    movel(pose_trans(stn7_plane, pose_trans(p[.109811488584, -1.023382701287, -.166619380160, .003048702642, -.008599620441, 2.442192581404], stn7_dr1_dwn_p_p)), a=0.1, v=0.05)
    # begin: URCap Program Node
    #   Source: Robotiq_Grippers, 1.8.13.22852, Robotiq Inc.
    #   Type: Greifer
    $ 1330 "Greifer offen (1)"
    if not(gripper_connected[0]):
      popup("Greifer 1 muss verbunden sein, um dieses Programm auszuführen.", "Keine Verbindung", False, True, True)
    end
    if not(rq_is_gripper_activated("1")):
      popup("Greifer 1 ist nicht aktiviert. Wechseln Sie zur Registerkarte Installation > Greifer, um ihn zu aktivieren und das Programm erneut auszuführen.", "Nicht aktiviert", False, True, True)
    end
    rq_set_pos_spd_for(0, 255, 0, "1")
    rq_wait_pos_spe_for_request(0, 255, 0, "1")
    rq_go_to("1")
    rq_wait("1")
    # end: URCap Program Node
    $ 1331 "stn7_dr1_up_p" "breakAfter"
    set_tcp(p[-3.0E-4,2.5E-4,0.1575,0.0,0.0,0.0])
    movel(pose_trans(stn7_plane, pose_trans(p[.109811488584, -1.023382701287, -.166619380160, .003048702642, -.008599620441, 2.442192581404], stn7_dr1_up_p_p)), a=0.1, v=0.05)
    # begin: URCap Program Node
    #   Source: Robotiq_Grippers, 1.8.13.22852, Robotiq Inc.
    #   Type: Greifer
    $ 1332 "Greifer geschlossen (1)"
    if not(gripper_connected[0]):
      popup("Greifer 1 muss verbunden sein, um dieses Programm auszuführen.", "Keine Verbindung", False, True, True)
    end
    if not(rq_is_gripper_activated("1")):
      popup("Greifer 1 ist nicht aktiviert. Wechseln Sie zur Registerkarte Installation > Greifer, um ihn zu aktivieren und das Programm erneut auszuführen.", "Nicht aktiviert", False, True, True)
    end
    rq_set_pos_spd_for(255, 255, 0, "1")
    rq_wait_pos_spe_for_request(255, 255, 0, "1")
    rq_go_to("1")
    rq_wait("1")
    # end: URCap Program Node
    $ 1333 "FahreAchse"
    $ 1334 "stn7_ld_apr_p" "breakAfter"
    set_tcp(p[-3.0E-4,2.5E-4,0.1575,0.0,0.0,0.0])
    movej(get_inverse_kin(pose_trans(stn7_plane, pose_trans(p[.109811488584, -1.023382701287, -.166619380160, .003048702642, -.008599620441, 2.442192581404], stn7_ld_apr_p_p)), qnear=stn7_ld_apr_p_q), a=2.443460952792061, v=1.7453292519943295)
    $ 1335 "FahreLinear"
    $ 1336 "stn7_ld_press_p" "breakAfter"
    set_tcp(p[-3.0E-4,2.5E-4,0.1575,0.0,0.0,0.0])
    movel(pose_trans(stn7_plane, pose_trans(p[.109811488584, -1.023382701287, -.166619380160, .003048702642, -.008599620441, 2.442192581404], stn7_ld_press_p_p)), a=0.6, v=0.1)
    $ 1337 "Warten: 1.0"
    sleep(1.0)
    $ 1338 "stn7_ld_apr_p" "breakAfter"
    set_tcp(p[-3.0E-4,2.5E-4,0.1575,0.0,0.0,0.0])
    movel(pose_trans(stn7_plane, pose_trans(p[.109811488584, -1.023382701287, -.166619380160, .003048702642, -.008599620441, 2.442192581404], stn7_ld_apr_p_p)), a=0.6, v=0.1)
    $ 1339 "qMast.set_init_alarm(7)"
    qMast.set_init_alarm(7)
    $ 1340 "FahreAchse"
    $ 1341 "stn7_home_p" "breakAfter"
    set_tcp(p[-3.0E-4,2.5E-4,0.1575,0.0,0.0,0.0])
    movej(get_inverse_kin(pose_trans(stn7_plane, pose_trans(p[.109811488584, -1.023382701287, -.166619380160, .003048702642, -.008599620441, 2.442192581404], stn7_home_p_p)), qnear=stn7_home_p_q), a=1.3962634015954636, v=1.0471975511965976)
  end
  def stn7_open_doors():
    $ 1342 "stn7_open_doors" "noBreak"
    $ 1343 "FahreAchse"
    $ 1345 "stn7_retrct1_p" "breakAfter"
    set_tcp(p[-3.0E-4,2.5E-4,0.1575,0.0,0.0,0.0])
    movej(get_inverse_kin(pose_trans(stn7_plane, pose_trans(p[.109811488584, -1.023382701287, -.166619380160, .003048702642, -.008599620441, 2.442192581404], stn7_retrct1_p_p)), qnear=stn7_retrct1_p_q), a=1.3962634015954636, v=1.0471975511965976)
    $ 1346 "stn7_dr1_up_p" "breakAfter"
    set_tcp(p[-3.0E-4,2.5E-4,0.1575,0.0,0.0,0.0])
    movej(get_inverse_kin(pose_trans(stn7_plane, pose_trans(p[.109811488584, -1.023382701287, -.166619380160, .003048702642, -.008599620441, 2.442192581404], stn7_dr1_up_p_p)), qnear=stn7_dr1_up_p_q), a=1.3962634015954636, v=1.0471975511965976)
    # begin: URCap Program Node
    #   Source: Robotiq_Grippers, 1.8.13.22852, Robotiq Inc.
    #   Type: Greifer
    $ 1347 "Greifer offen (1)"
    if not(gripper_connected[0]):
      popup("Greifer 1 muss verbunden sein, um dieses Programm auszuführen.", "Keine Verbindung", False, True, True)
    end
    if not(rq_is_gripper_activated("1")):
      popup("Greifer 1 ist nicht aktiviert. Wechseln Sie zur Registerkarte Installation > Greifer, um ihn zu aktivieren und das Programm erneut auszuführen.", "Nicht aktiviert", False, True, True)
    end
    rq_set_pos_spd_for(0, 255, 0, "1")
    rq_wait_pos_spe_for_request(0, 255, 0, "1")
    rq_go_to("1")
    rq_wait("1")
    # end: URCap Program Node
    $ 1348 "FahreLinear"
    $ 1349 "stn7_dr1_dwn_p" "breakAfter"
    set_tcp(p[-3.0E-4,2.5E-4,0.1575,0.0,0.0,0.0])
    movel(pose_trans(stn7_plane, pose_trans(p[.109811488584, -1.023382701287, -.166619380160, .003048702642, -.008599620441, 2.442192581404], stn7_dr1_dwn_p_p)), a=0.3, v=0.1)
    $ 1350 "stn7_dr1_open_p" "breakAfter"
    set_tcp(p[-3.0E-4,2.5E-4,0.1575,0.0,0.0,0.0])
    movel(pose_trans(stn7_plane, pose_trans(p[.109811488584, -1.023382701287, -.166619380160, .003048702642, -.008599620441, 2.442192581404], stn7_dr1_open_p_p)), a=0.3, v=0.1)
    $ 1351 "stn7_dr2_ohp1_p" "breakAfter"
    set_tcp(p[-3.0E-4,2.5E-4,0.1575,0.0,0.0,0.0])
    movel(pose_trans(stn7_plane, pose_trans(p[.109811488584, -1.023382701287, -.166619380160, .003048702642, -.008599620441, 2.442192581404], stn7_dr2_ohp1_p_p)), a=0.3, v=0.1)
    $ 1352 "FahreLinear"
    $ 1353 "stn7_dr2_up_p" "breakAfter"
    set_tcp(p[-3.0E-4,2.5E-4,0.1575,0.0,0.0,0.0])
    movel(pose_trans(stn7_plane, pose_trans(p[.109811488584, -1.023382701287, -.166619380160, .003048702642, -.008599620441, 2.442192581404], stn7_dr2_up_p_p)), a=0.3, v=0.1)
    $ 1354 "stn7_dr2_dwn_p" "breakAfter"
    set_tcp(p[-3.0E-4,2.5E-4,0.1575,0.0,0.0,0.0])
    movel(pose_trans(stn7_plane, pose_trans(p[.109811488584, -1.023382701287, -.166619380160, .003048702642, -.008599620441, 2.442192581404], stn7_dr2_dwn_p_p)), a=0.3, v=0.1)
    $ 1355 "stn7_dr2_open_p" "breakAfter"
    set_tcp(p[-3.0E-4,2.5E-4,0.1575,0.0,0.0,0.0])
    movel(pose_trans(stn7_plane, pose_trans(p[.109811488584, -1.023382701287, -.166619380160, .003048702642, -.008599620441, 2.442192581404], stn7_dr2_open_p_p)), a=0.3, v=0.1)
    $ 1356 "stn7_dr2_ohp1_p" "breakAfter"
    set_tcp(p[-3.0E-4,2.5E-4,0.1575,0.0,0.0,0.0])
    movel(pose_trans(stn7_plane, pose_trans(p[.109811488584, -1.023382701287, -.166619380160, .003048702642, -.008599620441, 2.442192581404], stn7_dr2_ohp1_p_p)), a=0.3, v=0.1)
    # begin: URCap Program Node
    #   Source: Robotiq_Grippers, 1.8.13.22852, Robotiq Inc.
    #   Type: Greifer
    $ 1357 "Greifer geschlossen (1)"
    if not(gripper_connected[0]):
      popup("Greifer 1 muss verbunden sein, um dieses Programm auszuführen.", "Keine Verbindung", False, True, True)
    end
    if not(rq_is_gripper_activated("1")):
      popup("Greifer 1 ist nicht aktiviert. Wechseln Sie zur Registerkarte Installation > Greifer, um ihn zu aktivieren und das Programm erneut auszuführen.", "Nicht aktiviert", False, True, True)
    end
    rq_set_pos_spd_for(255, 255, 0, "1")
    rq_wait_pos_spe_for_request(255, 255, 0, "1")
    rq_go_to("1")
    rq_wait("1")
    # end: URCap Program Node
    $ 1358 "FahreAchse"
    $ 1359 "stn7_home_p" "breakAfter"
    set_tcp(p[-3.0E-4,2.5E-4,0.1575,0.0,0.0,0.0])
    movej(get_inverse_kin(pose_trans(stn7_plane, pose_trans(p[.109811488584, -1.023382701287, -.166619380160, .003048702642, -.008599620441, 2.442192581404], stn7_home_p_p)), qnear=stn7_home_p_q), a=1.3962634015954636, v=1.0471975511965976)
  end
  def stn7_close_doors():
    $ 1360 "stn7_close_doors" "noBreak"
    # begin: URCap Program Node
    #   Source: Robotiq_Grippers, 1.8.13.22852, Robotiq Inc.
    #   Type: Greifer
    $ 1361 "Greifer geschlossen (1)"
    if not(gripper_connected[0]):
      popup("Greifer 1 muss verbunden sein, um dieses Programm auszuführen.", "Keine Verbindung", False, True, True)
    end
    if not(rq_is_gripper_activated("1")):
      popup("Greifer 1 ist nicht aktiviert. Wechseln Sie zur Registerkarte Installation > Greifer, um ihn zu aktivieren und das Programm erneut auszuführen.", "Nicht aktiviert", False, True, True)
    end
    rq_set_pos_spd_for(255, 128, 255, "1")
    rq_wait_pos_spe_for_request(255, 128, 255, "1")
    rq_go_to("1")
    rq_wait("1")
    # end: URCap Program Node
    $ 1362 "FahreAchse"
    $ 1363 "stn7_home_p" "breakAfter"
    set_tcp(p[-3.0E-4,2.5E-4,0.1575,0.0,0.0,0.0])
    movej(get_inverse_kin(pose_trans(stn7_plane, pose_trans(p[.109811488584, -1.023382701287, -.166619380160, .003048702642, -.008599620441, 2.442192581404], stn7_home_p_p)), qnear=stn7_home_p_q), a=1.3962634015954636, v=1.0471975511965976, r=0.1)
    $ 1364 "stn7_apr1_p" "breakAfter"
    set_tcp(p[-3.0E-4,2.5E-4,0.1575,0.0,0.0,0.0])
    movej(get_inverse_kin(pose_trans(stn7_plane, pose_trans(p[.109811488584, -1.023382701287, -.166619380160, .003048702642, -.008599620441, 2.442192581404], stn7_apr1_p_p)), qnear=stn7_apr1_p_q), a=1.3962634015954636, v=1.0471975511965976)
    $ 1365 "FahreLinear"
    $ 1366 "stn7_push1_p" "breakAfter"
    set_tcp(p[-3.0E-4,2.5E-4,0.1575,0.0,0.0,0.0])
    movel(pose_trans(stn7_plane, pose_trans(p[.109811488584, -1.023382701287, -.166619380160, .003048702642, -.008599620441, 2.442192581404], stn7_push1_p_p)), a=0.5, v=0.1)
    $ 1367 "stn7_apr1_p" "breakAfter"
    set_tcp(p[-3.0E-4,2.5E-4,0.1575,0.0,0.0,0.0])
    movel(pose_trans(stn7_plane, pose_trans(p[.109811488584, -1.023382701287, -.166619380160, .003048702642, -.008599620441, 2.442192581404], stn7_apr1_p_p)), a=1.2, v=0.25)
    $ 1368 "stn7_apr2_p" "breakAfter"
    set_tcp(p[-3.0E-4,2.5E-4,0.1575,0.0,0.0,0.0])
    movel(pose_trans(stn7_plane, pose_trans(p[.109811488584, -1.023382701287, -.166619380160, .003048702642, -.008599620441, 2.442192581404], stn7_apr2_p_p)), a=1.2, v=0.25)
    $ 1369 "stn7_push2_p" "breakAfter"
    set_tcp(p[-3.0E-4,2.5E-4,0.1575,0.0,0.0,0.0])
    movel(pose_trans(stn7_plane, pose_trans(p[.109811488584, -1.023382701287, -.166619380160, .003048702642, -.008599620441, 2.442192581404], stn7_push2_p_p)), a=0.5, v=0.1)
    $ 1370 "stn7_dr2_bk_p" "breakAfter"
    set_tcp(p[-3.0E-4,2.5E-4,0.1575,0.0,0.0,0.0])
    movel(pose_trans(stn7_plane, pose_trans(p[.109811488584, -1.023382701287, -.166619380160, .003048702642, -.008599620441, 2.442192581404], stn7_dr2_bk_p_p)), a=1.2, v=0.25)
  end
  def stn7_check_doors():
    $ 1371 "stn7_check_doors" "noBreak"
    $ 1372 "Schleife"
    while (True):
      $ 1373 "stn7_door_1_ok≔get_digital_in(2)"
      global stn7_door_1_ok=get_digital_in(2)
      $ 1374 "If stn7_door_1_ok ≟  False "
      if (stn7_door_1_ok  ==    False  ):
        $ 1376 "Meldung"
        popup(str_cat("",stn7_skype_msg), "Fehler", False, True, blocking=False)
        halt
      else:
        $ 1377 "Else" "noBreak"
        $ 1378 "stn7_door_2_ok≔get_digital_in(0)"
        global stn7_door_2_ok=get_digital_in(0)
        $ 1379 "If stn7_door_2_ok ≟  False "
        if (stn7_door_2_ok  ==    False  ):
          $ 1381 "Meldung"
          popup(str_cat("",stn7_skype_msg), "Fehler", False, True, blocking=False)
          halt
        else:
          $ 1382 "Else" "noBreak"
          $ 1383 "break"
          break
        end
      end
    end
  end
  def stn9_decap():
    $ 1384 "stn9_decap" "noBreak"
    $ 1385 "FahreAchse"
    $ 1386 "stn9_dcap_apr_p" "breakAfter"
    set_tcp(p[-3.0E-4,2.5E-4,0.1575,0.0,0.0,0.0])
    movej(get_inverse_kin(pose_trans(stn6_plane, pose_trans(p[.776557109756, -.878329076792, .250244777977, -.001605684562, .009314448336, 1.565629725105], stn9_dcap_apr_p_p)), qnear=stn9_dcap_apr_p_q), a=2.792526803190927, v=2.0943951023931953)
    $ 1387 "Einstellen Decap=Ein"
    set_standard_digital_out(2, True)
    $ 1388 "FahreLinear"
    $ 1389 "stn9_lv_tb_p" "breakAfter"
    set_tcp(p[-3.0E-4,2.5E-4,0.1575,0.0,0.0,0.0])
    movel(pose_trans(stn6_plane, pose_trans(p[.776557109756, -.878329076792, .250244777977, -.001605684562, .009314448336, 1.565629725105], stn9_lv_tb_p_p)), a=0.6, v=0.12)
    # begin: URCap Program Node
    #   Source: Robotiq_Grippers, 1.8.13.22852, Robotiq Inc.
    #   Type: Greifer
    $ 1390 "Greiferbewegung65% (1)"
    if not(gripper_connected[0]):
      popup("Greifer 1 muss verbunden sein, um dieses Programm auszuführen.", "Keine Verbindung", False, True, True)
    end
    if not(rq_is_gripper_activated("1")):
      popup("Greifer 1 ist nicht aktiviert. Wechseln Sie zur Registerkarte Installation > Greifer, um ihn zu aktivieren und das Programm erneut auszuführen.", "Nicht aktiviert", False, True, True)
    end
    rq_set_pos_spd_for(166, 51, 0, "1")
    rq_wait_pos_spe_for_request(166, 51, 0, "1")
    rq_go_to("1")
    rq_wait("1")
    # end: URCap Program Node
    $ 1391 "Warten: 0.5"
    sleep(0.5)
    $ 1392 "Einstellen Decap=Aus"
    set_standard_digital_out(2, False)
    $ 1393 "FahreAchse"
    $ 1394 "stn9_hold_dcp_p" "breakAfter"
    set_tcp(p[-3.0E-4,2.5E-4,0.1575,0.0,0.0,0.0])
    movej(get_inverse_kin(pose_trans(stn6_plane, pose_trans(p[.776557109756, -.878329076792, .250244777977, -.001605684562, .009314448336, 1.565629725105], stn9_hold_dcp_p_p)), qnear=stn9_hold_dcp_p_q), a=20.943951023931955, v=3.141592653589793)
    # begin: URCap Program Node
    #   Source: Robotiq_Grippers, 1.8.13.22852, Robotiq Inc.
    #   Type: Greifer
    $ 1395 "Greifer geschlossen (1)"
    if not(gripper_connected[0]):
      popup("Greifer 1 muss verbunden sein, um dieses Programm auszuführen.", "Keine Verbindung", False, True, True)
    end
    if not(rq_is_gripper_activated("1")):
      popup("Greifer 1 ist nicht aktiviert. Wechseln Sie zur Registerkarte Installation > Greifer, um ihn zu aktivieren und das Programm erneut auszuführen.", "Nicht aktiviert", False, True, True)
    end
    rq_set_pos_spd_for(255, 128, 128, "1")
    rq_wait_pos_spe_for_request(255, 128, 128, "1")
    rq_go_to("1")
    rq_wait("1")
    # end: URCap Program Node
    $ 1396 "FahreAchse"
    $ 1397 "stn9_dcap_up_p" "breakAfter"
    set_tcp(p[-3.0E-4,2.5E-4,0.1575,0.0,0.0,0.0])
    movej(get_inverse_kin(pose_trans(stn6_plane, pose_trans(p[.776557109756, -.878329076792, .250244777977, -.001605684562, .009314448336, 1.565629725105], stn9_dcap_up_p_p)), qnear=stn9_dcap_up_p_q), a=2.792526803190927, v=1.0471975511965976)
    $ 1398 "FahreLinear"
    $ 1399 "stn9_dcap_hlp_p" "breakAfter"
    set_tcp(p[-3.0E-4,2.5E-4,0.1575,0.0,0.0,0.0])
    movel(pose_trans(stn6_plane, pose_trans(p[.776557109756, -.878329076792, .250244777977, -.001605684562, .009314448336, 1.565629725105], stn9_dcap_hlp_p_p)), a=0.8, v=0.5)
    $ 1400 "FahreAchse"
    $ 1401 "stn9_dcap_apr_p" "breakAfter"
    set_tcp(p[-3.0E-4,2.5E-4,0.1575,0.0,0.0,0.0])
    movej(get_inverse_kin(pose_trans(stn6_plane, pose_trans(p[.776557109756, -.878329076792, .250244777977, -.001605684562, .009314448336, 1.565629725105], stn9_dcap_apr_p_p)), qnear=stn9_dcap_apr_p_q), a=20.943951023931955, v=3.141592653589793)
    $ 1402 "FahreAchse"
    $ 1403 "stn9_bin_apr_p" "breakAfter"
    set_tcp(p[-3.0E-4,2.5E-4,0.1575,0.0,0.0,0.0])
    movej(get_inverse_kin(pose_trans(stn6_plane, pose_trans(p[.776557109756, -.878329076792, .250244777977, -.001605684562, .009314448336, 1.565629725105], stn9_bin_apr_p_p)), qnear=stn9_bin_apr_p_q), a=3.490658503988659, v=1.0471975511965976, r=0.005)
    $ 1404 "stn9_lv_cap_p" "breakAfter"
    set_tcp(p[-3.0E-4,2.5E-4,0.1575,0.0,0.0,0.0])
    movej(get_inverse_kin(pose_trans(stn6_plane, pose_trans(p[.776557109756, -.878329076792, .250244777977, -.001605684562, .009314448336, 1.565629725105], stn9_lv_cap_p_p)), qnear=stn9_lv_cap_p_q), a=3.490658503988659, v=1.0471975511965976)
    # begin: URCap Program Node
    #   Source: Robotiq_Grippers, 1.8.13.22852, Robotiq Inc.
    #   Type: Greifer
    $ 1405 "Greiferbewegung50% (1)"
    if not(gripper_connected[0]):
      popup("Greifer 1 muss verbunden sein, um dieses Programm auszuführen.", "Keine Verbindung", False, True, True)
    end
    if not(rq_is_gripper_activated("1")):
      popup("Greifer 1 ist nicht aktiviert. Wechseln Sie zur Registerkarte Installation > Greifer, um ihn zu aktivieren und das Programm erneut auszuführen.", "Nicht aktiviert", False, True, True)
    end
    rq_set_pos_spd_for(128, 255, 0, "1")
    rq_wait_pos_spe_for_request(128, 255, 0, "1")
    rq_go_to("1")
    rq_wait("1")
    # end: URCap Program Node
    # begin: URCap Program Node
    #   Source: Robotiq_Grippers, 1.8.13.22852, Robotiq Inc.
    #   Type: Greifer
    $ 1406 "Greifer geschlossen (1)"
    if not(gripper_connected[0]):
      popup("Greifer 1 muss verbunden sein, um dieses Programm auszuführen.", "Keine Verbindung", False, True, True)
    end
    if not(rq_is_gripper_activated("1")):
      popup("Greifer 1 ist nicht aktiviert. Wechseln Sie zur Registerkarte Installation > Greifer, um ihn zu aktivieren und das Programm erneut auszuführen.", "Nicht aktiviert", False, True, True)
    end
    rq_set_pos_spd_for(255, 64, 0, "1")
    rq_wait_pos_spe_for_request(255, 64, 0, "1")
    rq_go_to("1")
    rq_wait("1")
    # end: URCap Program Node
    # begin: URCap Program Node
    #   Source: Robotiq_Grippers, 1.8.13.22852, Robotiq Inc.
    #   Type: Greifer
    $ 1407 "Greiferbewegung50% (1)"
    if not(gripper_connected[0]):
      popup("Greifer 1 muss verbunden sein, um dieses Programm auszuführen.", "Keine Verbindung", False, True, True)
    end
    if not(rq_is_gripper_activated("1")):
      popup("Greifer 1 ist nicht aktiviert. Wechseln Sie zur Registerkarte Installation > Greifer, um ihn zu aktivieren und das Programm erneut auszuführen.", "Nicht aktiviert", False, True, True)
    end
    rq_set_pos_spd_for(128, 255, 0, "1")
    rq_wait_pos_spe_for_request(128, 255, 0, "1")
    rq_go_to("1")
    rq_wait("1")
    # end: URCap Program Node
    $ 1408 "FahreAchse"
    $ 1409 "stn9_bin_apr_p" "breakAfter"
    set_tcp(p[-3.0E-4,2.5E-4,0.1575,0.0,0.0,0.0])
    movej(get_inverse_kin(pose_trans(stn6_plane, pose_trans(p[.776557109756, -.878329076792, .250244777977, -.001605684562, .009314448336, 1.565629725105], stn9_bin_apr_p_p)), qnear=stn9_bin_apr_p_q), a=3.490658503988659, v=1.0471975511965976, r=0.005)
    $ 1410 "stn9_dcap_apr_p" "breakAfter"
    set_tcp(p[-3.0E-4,2.5E-4,0.1575,0.0,0.0,0.0])
    movej(get_inverse_kin(pose_trans(stn6_plane, pose_trans(p[.776557109756, -.878329076792, .250244777977, -.001605684562, .009314448336, 1.565629725105], stn9_dcap_apr_p_p)), qnear=stn9_dcap_apr_p_q), a=3.490658503988659, v=1.0471975511965976)
    # begin: URCap Program Node
    #   Source: Robotiq_Grippers, 1.8.13.22852, Robotiq Inc.
    #   Type: Greifer
    $ 1411 "Greifer offen (1)"
    if not(gripper_connected[0]):
      popup("Greifer 1 muss verbunden sein, um dieses Programm auszuführen.", "Keine Verbindung", False, True, True)
    end
    if not(rq_is_gripper_activated("1")):
      popup("Greifer 1 ist nicht aktiviert. Wechseln Sie zur Registerkarte Installation > Greifer, um ihn zu aktivieren und das Programm erneut auszuführen.", "Nicht aktiviert", False, True, True)
    end
    rq_set_pos_spd_for(0, 255, 0, "1")
    rq_wait_pos_spe_for_request(0, 255, 0, "1")
    rq_go_to("1")
    rq_wait("1")
    # end: URCap Program Node
    $ 1412 "FahreLinear"
    $ 1413 "stn9_hold_cap_p" "breakAfter"
    set_tcp(p[-3.0E-4,2.5E-4,0.1575,0.0,0.0,0.0])
    movel(pose_trans(stn6_plane, pose_trans(p[.776557109756, -.878329076792, .250244777977, -.001605684562, .009314448336, 1.565629725105], stn9_hold_cap_p_p)), a=0.8, v=0.25)
    # begin: URCap Program Node
    #   Source: Robotiq_Grippers, 1.8.13.22852, Robotiq Inc.
    #   Type: Greifer
    $ 1414 "Greifer geschlossen (1)"
    if not(gripper_connected[0]):
      popup("Greifer 1 muss verbunden sein, um dieses Programm auszuführen.", "Keine Verbindung", False, True, True)
    end
    if not(rq_is_gripper_activated("1")):
      popup("Greifer 1 ist nicht aktiviert. Wechseln Sie zur Registerkarte Installation > Greifer, um ihn zu aktivieren und das Programm erneut auszuführen.", "Nicht aktiviert", False, True, True)
    end
    rq_set_pos_spd_for(255, 128, 51, "1")
    rq_wait_pos_spe_for_request(255, 128, 51, "1")
    rq_go_to("1")
    rq_wait("1")
    # end: URCap Program Node
    $ 1415 "Einstellen Decap=Ein"
    set_standard_digital_out(2, True)
    $ 1416 "FahreLinear"
    $ 1417 "stn9_dcap_apr_p" "breakAfter"
    set_tcp(p[-3.0E-4,2.5E-4,0.1575,0.0,0.0,0.0])
    movel(pose_trans(stn6_plane, pose_trans(p[.776557109756, -.878329076792, .250244777977, -.001605684562, .009314448336, 1.565629725105], stn9_dcap_apr_p_p)), a=1.2, v=0.25)
  end
  def stn11_open_archiv():
    $ 1418 "stn11_open_archiv" "noBreak"
    # begin: URCap Program Node
    #   Source: Robotiq_Grippers, 1.8.13.22852, Robotiq Inc.
    #   Type: Greifer
    $ 1419 "Greifer geschlossen (1)"
    if not(gripper_connected[0]):
      popup("Greifer 1 muss verbunden sein, um dieses Programm auszuführen.", "Keine Verbindung", False, True, True)
    end
    if not(rq_is_gripper_activated("1")):
      popup("Greifer 1 ist nicht aktiviert. Wechseln Sie zur Registerkarte Installation > Greifer, um ihn zu aktivieren und das Programm erneut auszuführen.", "Nicht aktiviert", False, True, True)
    end
    rq_set_pos_spd_for(255, 255, 255, "1")
    rq_wait_pos_spe_for_request(255, 255, 255, "1")
    rq_go_to("1")
    rq_wait("1")
    # end: URCap Program Node
    $ 1420 "FahreAchse"
    $ 1421 "stn11_home_p" "breakAfter"
    set_tcp(p[-3.0E-4,2.5E-4,0.1575,0.0,0.0,0.0])
    movej(get_inverse_kin(pose_trans(stn6_plane, pose_trans(p[.776557109756, -.878329076792, .250244777977, -.001605684562, .009314448336, 1.565629725105], stn11_home_p_p)), qnear=stn11_home_p_q), a=1.3962634015954636, v=1.0471975511965976)
    $ 1422 "FahreLinear"
    $ 1423 "stn11_hlp_up_p" "breakAfter"
    set_tcp(p[-3.0E-4,2.5E-4,0.1575,0.0,0.0,0.0])
    movel(pose_trans(stn6_plane, pose_trans(p[.776557109756, -.878329076792, .250244777977, -.001605684562, .009314448336, 1.565629725105], stn11_hlp_up_p_p)), a=1.2, v=0.25)
    $ 1424 "stn11_clo_apr_p" "breakAfter"
    set_tcp(p[-3.0E-4,2.5E-4,0.1575,0.0,0.0,0.0])
    movel(pose_trans(stn6_plane, pose_trans(p[.776557109756, -.878329076792, .250244777977, -.001605684562, .009314448336, 1.565629725105], stn11_clo_apr_p_p)), a=1.2, v=0.25)
    $ 1425 "stn11_close_p" "breakAfter"
    set_tcp(p[-3.0E-4,2.5E-4,0.1575,0.0,0.0,0.0])
    movel(pose_trans(stn6_plane, pose_trans(p[.776557109756, -.878329076792, .250244777977, -.001605684562, .009314448336, 1.565629725105], stn11_close_p_p)), a=0.5, v=0.1)
    $ 1426 "stn11_clo_up_p" "breakAfter"
    set_tcp(p[-3.0E-4,2.5E-4,0.1575,0.0,0.0,0.0])
    movel(pose_trans(stn6_plane, pose_trans(p[.776557109756, -.878329076792, .250244777977, -.001605684562, .009314448336, 1.565629725105], stn11_clo_up_p_p)), a=1.2, v=0.25)
    $ 1427 "stn11_clo_up2_p" "breakAfter"
    set_tcp(p[-3.0E-4,2.5E-4,0.1575,0.0,0.0,0.0])
    movel(pose_trans(stn6_plane, pose_trans(p[.776557109756, -.878329076792, .250244777977, -.001605684562, .009314448336, 1.565629725105], stn11_clo_up2_p_p)), a=1.2, v=0.25)
    # begin: URCap Program Node
    #   Source: Robotiq_Grippers, 1.8.13.22852, Robotiq Inc.
    #   Type: Greifer
    $ 1428 "Greifer offen (1)"
    if not(gripper_connected[0]):
      popup("Greifer 1 muss verbunden sein, um dieses Programm auszuführen.", "Keine Verbindung", False, True, True)
    end
    if not(rq_is_gripper_activated("1")):
      popup("Greifer 1 ist nicht aktiviert. Wechseln Sie zur Registerkarte Installation > Greifer, um ihn zu aktivieren und das Programm erneut auszuführen.", "Nicht aktiviert", False, True, True)
    end
    rq_set_pos_spd_for(0, 255, 255, "1")
    rq_wait_pos_spe_for_request(0, 255, 255, "1")
    rq_go_to("1")
    rq_wait("1")
    # end: URCap Program Node
    $ 1429 "stn11_opn_apr_p" "breakAfter"
    set_tcp(p[-3.0E-4,2.5E-4,0.1575,0.0,0.0,0.0])
    movel(pose_trans(stn6_plane, pose_trans(p[.776557109756, -.878329076792, .250244777977, -.001605684562, .009314448336, 1.565629725105], stn11_opn_apr_p_p)), a=1.2, v=0.25)
    $ 1430 "stn11_opn_p" "breakAfter"
    set_tcp(p[-3.0E-4,2.5E-4,0.1575,0.0,0.0,0.0])
    movel(pose_trans(stn6_plane, pose_trans(p[.776557109756, -.878329076792, .250244777977, -.001605684562, .009314448336, 1.565629725105], stn11_opn_p_p)), a=0.5, v=0.1)
    $ 1431 "stn11_opn_up_p" "breakAfter"
    set_tcp(p[-3.0E-4,2.5E-4,0.1575,0.0,0.0,0.0])
    movel(pose_trans(stn6_plane, pose_trans(p[.776557109756, -.878329076792, .250244777977, -.001605684562, .009314448336, 1.565629725105], stn11_opn_up_p_p)), a=1.2, v=0.25)
    # begin: URCap Program Node
    #   Source: Robotiq_Grippers, 1.8.13.22852, Robotiq Inc.
    #   Type: Greifer
    $ 1432 "Greifer geschlossen (1)"
    if not(gripper_connected[0]):
      popup("Greifer 1 muss verbunden sein, um dieses Programm auszuführen.", "Keine Verbindung", False, True, True)
    end
    if not(rq_is_gripper_activated("1")):
      popup("Greifer 1 ist nicht aktiviert. Wechseln Sie zur Registerkarte Installation > Greifer, um ihn zu aktivieren und das Programm erneut auszuführen.", "Nicht aktiviert", False, True, True)
    end
    rq_set_pos_spd_for(255, 255, 255, "1")
    rq_wait_pos_spe_for_request(255, 255, 255, "1")
    rq_go_to("1")
    rq_wait("1")
    # end: URCap Program Node
    $ 1433 "FahreAchse"
    $ 1434 "stn11_home_p" "breakAfter"
    set_tcp(p[-3.0E-4,2.5E-4,0.1575,0.0,0.0,0.0])
    movej(get_inverse_kin(pose_trans(stn6_plane, pose_trans(p[.776557109756, -.878329076792, .250244777977, -.001605684562, .009314448336, 1.565629725105], stn11_home_p_p)), qnear=stn11_home_p_q), a=1.3962634015954636, v=1.0471975511965976)
  end
  $ 1 "VorStart"
  $ 2 "stn3_ok_popup≔ True "
  global stn3_ok_popup=  True
  $ 3 "stn3_cros_popup≔ True "
  global stn3_cros_popup=  True
  $ 4 "qMast≔rpc_factory('xmlrpc','http://192.168.20.222:9095')"
  global qMast=rpc_factory("xmlrpc","http://192.168.20.222:9095")
  $ 6 "all_machines_on≔ False "
  global all_machines_on=  False
  $ 7 "bc_2_check≔ True "
  global bc_2_check=  True
  $ 8 "init_qMast≔ True "
  global init_qMast=  True
  $ 9 "start_ping≔ False "
  global start_ping=  False
  $ 10 "jobDone≔ False "
  global jobDone=  False
  $ 11 "jobID≔-1"
  global jobID=-1
  $ 12 "Teach≔ False "
  global Teach=  False
  $ 13 "goToHome≔ True "
  global goToHome=  True
  $ 14 "moveToHome≔ False "
  global moveToHome=  False
  $ 15 "stn2_ini_chk_rk≔ True "
  global stn2_ini_chk_rk=  True
  $ 16 "cam2_angle≔10"
  global cam2_angle=10
  $ 17 "cam2_angle2≔5"
  global cam2_angle2=5
  $ 18 "stn1_rows≔5"
  global stn1_rows=5
  $ 19 "stn1_cols≔8"
  global stn1_cols=8
  $ 20 "stn1_pick_z≔123"
  global stn1_pick_z=123
  $ 21 "stn3_total_locs≔10"
  global stn3_total_locs=10
  $ 22 "stn3_place_z≔21"
  global stn3_place_z=21
  $ 23 "stn3_rot_z≔60"
  global stn3_rot_z=60
  $ 24 "stn3_pick_z≔81"
  global stn3_pick_z=81
  $ 25 "stn2_pk_rk_z≔136"
  global stn2_pk_rk_z=136
  $ 26 "stn2_rk_chk_y≔64"
  global stn2_rk_chk_y=64
  $ 27 "stn4_loop_count≔0"
  global stn4_loop_count=0
  $ 28 "stn5_pick_tb_z≔124"
  global stn5_pick_tb_z=124
  $ 29 "stn5_place_tb_z≔120"
  global stn5_place_tb_z=120
  $ 30 "stn5_place_rk_z≔121"
  global stn5_place_rk_z=121
  $ 31 "stn5_pick_rk_z≔121"
  global stn5_pick_rk_z=121
  $ 32 "stn5_pick_cw_z≔120"
  global stn5_pick_cw_z=120
  $ 33 "stn5_place_cw_z≔118"
  global stn5_place_cw_z=118
  $ 34 "stn5_rows_parnt≔4"
  global stn5_rows_parnt=4
  $ 35 "stn5_cols_parnt≔2"
  global stn5_cols_parnt=2
  $ 36 "stn5_rows_child≔3"
  global stn5_rows_child=3
  $ 37 "stn5_cols_child≔3"
  global stn5_cols_child=3
  $ 38 "stn6_pick_z≔254"
  global stn6_pick_z=254
  $ 39 "stn6_place_z≔250"
  global stn6_place_z=250
  $ 40 "stn7_rows_parnt≔1"
  global stn7_rows_parnt=1
  $ 41 "stn7_cols_parnt≔2"
  global stn7_cols_parnt=2
  $ 42 "stn7_rows_child≔2"
  global stn7_rows_child=2
  $ 43 "stn7_cols_child≔5"
  global stn7_cols_child=5
  $ 44 "stn7_place_z≔199"
  global stn7_place_z=199
  $ 45 "stn7_pick_z≔204"
  global stn7_pick_z=204
  $ 46 "stn7_skype_msg≔'Sysmex Schubladenpos. manuell veraendert. Roboter bitte neu starten. Herzliche Gruesse Markus Praus'"
  global stn7_skype_msg="Sysmex Schubladenpos. manuell veraendert. Roboter bitte neu starten. Herzliche Gruesse Markus Praus"
  $ 47 "stn10_place_z≔175"
  global stn10_place_z=175
  $ 48 "stn10_skype_ful≔'Fehlerstaender ist full. Bitte roboter neu starten'"
  global stn10_skype_ful="Fehlerstaender ist full. Bitte roboter neu starten"
  $ 49 "stn11_place_z≔175"
  global stn11_place_z=175
  $ 50 "stn11_skype_msg≔'Bitte Archiv schublade offnen. Roboter bitte neu starten. Herzliche Gruesse Mrkus Praus'"
  global stn11_skype_msg="Bitte Archiv schublade offnen. Roboter bitte neu starten. Herzliche Gruesse Mrkus Praus"
  $ 51 "stn11_skype_ful≔'Archivstaender ist full. Bitte roboter neu starten'"
  global stn11_skype_ful="Archivstaender ist full. Bitte roboter neu starten"
  $ 52 "stn14_tb_rot_z≔70"
  global stn14_tb_rot_z=70
  $ 53 "stn14_tb_pl_z≔38"
  global stn14_tb_pl_z=38
  $ 54 "stn14_push_z≔70"
  global stn14_push_z=70
  $ 55 "stn14_pl_rk_z≔141"
  global stn14_pl_rk_z=141
  $ 56 "stn15_place_z≔175"
  global stn15_place_z=175
  $ 57 "stn15_pick_z≔178"
  global stn15_pick_z=178
  $ 58 "archiv_opened≔ False "
  global archiv_opened=  False
  $ 59 "Test≔ False "
  global Test=  False
  $ 1435 "Thread_1"
  thread Thread_1():
    while (True):
      $ 1436 "sync()"
      sync()
      $ 1437 "If jobDone≟ True "
      if (jobDone ==   True  ):
        $ 1438 "jobArr≔qMast.get_job()"
        global jobArr=qMast.get_job()
        $ 1439 "jobID≔jobArr[0]"
        global jobID=jobArr[0]
        $ 1440 "If jobID ≠ 0"
        if (jobID  !=  0):
          $ 1441 "jobDone≔ False "
          global jobDone=  False
        end
      end
    end
  end
  threadId_Thread_1 = run Thread_1()
  $ 1442 "Thread_2"
  thread Thread_2():
    while (True):
      $ 1443 "sync()"
      sync()
      $ 1444 "Warten: 0.1"
      sleep(0.1)
      $ 1445 "If start_ping ≟  True "
      if (start_ping  ==    True  ):
        $ 1446 "qMast.ping()"
        qMast.ping()
      end
    end
  end
  threadId_Thread_2 = run Thread_2()
  while (True):
    $ 60 "Roboterprogramm"
    $ 61 "sync()"
    sync()
    $ 62 "If goToHome ≟  True "
    if (goToHome  ==    True  ):
      $ 63 "FahreAchse"
      $ 64 "home_p" "breakAfter"
      set_tcp(p[-3.0E-4,2.5E-4,0.1575,0.0,0.0,0.0])
      movej(get_inverse_kin(pose_trans(stn1_plane, pose_trans(p[.053539610991, -.984987293150, -.024848236577, .000189536594, .000276418508, 3.136265531618], home_p_p)), qnear=home_p_q), a=1.3962634015954636, v=1.0471975511965976)
      $ 65 "stn1_home_p" "breakAfter"
      set_tcp(p[-3.0E-4,2.5E-4,0.1575,0.0,0.0,0.0])
      movej(get_inverse_kin(pose_trans(stn1_plane, pose_trans(p[.053539610991, -.984987293150, -.024848236577, .000189536594, .000276418508, 3.136265531618], stn1_home_p_p)), qnear=stn1_home_p_q), a=1.3962634015954636, v=1.0471975511965976)
      $ 66 "goToHome≔ False "
      global goToHome=  False
    end
    $ 67 "If Teach≟ True "
    if (Teach ==   True  ):
      $ 68 "'Station 1 Reference Positions'"
      # 'Station 1 Reference Positions'
      $ 69 "FahreAchse"
      $ 70 "stn1_home_p" "breakAfter"
      set_tcp(p[-3.0E-4,2.5E-4,0.1575,0.0,0.0,0.0])
      movej(get_inverse_kin(pose_trans(stn1_plane, pose_trans(p[.053539610991, -.984987293150, -.024848236577, .000189536594, .000276418508, 3.136265531618], stn1_home_p_p)), qnear=stn1_home_p_q), a=1.3962634015954636, v=1.0471975511965976)
      $ 71 "stn1_help_p" "breakAfter"
      set_tcp(p[-3.0E-4,2.5E-4,0.1575,0.0,0.0,0.0])
      movej(get_inverse_kin(pose_trans(stn1_plane, pose_trans(p[.053539610991, -.984987293150, -.024848236577, .000189536594, .000276418508, 3.136265531618], stn1_help_p_p)), qnear=stn1_help_p_q), a=1.3962634015954636, v=1.0471975511965976)
      $ 72 "stn1_help2_p" "breakAfter"
      set_tcp(p[-3.0E-4,2.5E-4,0.1575,0.0,0.0,0.0])
      movej(get_inverse_kin(pose_trans(stn1_plane, pose_trans(p[.053539610991, -.984987293150, -.024848236577, .000189536594, .000276418508, 3.136265531618], stn1_help2_p_p)), qnear=stn1_help2_p_q), a=1.3962634015954636, v=1.0471975511965976)
      $ 73 "stn1_ref_1_p" "breakAfter"
      set_tcp(p[-3.0E-4,2.5E-4,0.1575,0.0,0.0,0.0])
      movej(get_inverse_kin(pose_trans(stn1_plane, pose_trans(p[.053539610991, -.984987293150, -.024848236577, .000189536594, .000276418508, 3.136265531618], stn1_ref_1_p_p)), qnear=stn1_ref_1_p_q), a=1.3962634015954636, v=1.0471975511965976)
      $ 74 "stn1_ref_2_p" "breakAfter"
      set_tcp(p[-3.0E-4,2.5E-4,0.1575,0.0,0.0,0.0])
      movej(get_inverse_kin(pose_trans(stn1_plane, pose_trans(p[.053539610991, -.984987293150, -.024848236577, .000189536594, .000276418508, 3.136265531618], stn1_ref_2_p_p)), qnear=stn1_ref_2_p_q), a=1.3962634015954636, v=1.0471975511965976)
      $ 75 "stn1_ref_3_p" "breakAfter"
      set_tcp(p[-3.0E-4,2.5E-4,0.1575,0.0,0.0,0.0])
      movej(get_inverse_kin(pose_trans(stn1_plane, pose_trans(p[.053539610991, -.984987293150, -.024848236577, .000189536594, .000276418508, 3.136265531618], stn1_ref_3_p_p)), qnear=stn1_ref_3_p_q), a=1.3962634015954636, v=1.0471975511965976)
      $ 76 "'Station 2 Reference Positions'"
      # 'Station 2 Reference Positions'
      $ 77 "FahreAchse"
      $ 78 "stn2_home_p" "breakAfter"
      set_tcp(p[-3.0E-4,2.5E-4,0.1575,0.0,0.0,0.0])
      movej(get_inverse_kin(pose_trans(stn2_plane, pose_trans(p[.137500819741, -.686313800478, .149495066037, -.008721928164, .022313263547, 3.131433712319], stn2_home_p_p)), qnear=stn2_home_p_q), a=1.3962634015954636, v=1.0471975511965976)
      $ 79 "stn2_ref_1_p" "breakAfter"
      set_tcp(p[-3.0E-4,2.5E-4,0.1575,0.0,0.0,0.0])
      movej(get_inverse_kin(pose_trans(stn2_plane, pose_trans(p[.137500819741, -.686313800478, .149495066037, -.008721928164, .022313263547, 3.131433712319], stn2_ref_1_p_p)), qnear=stn2_ref_1_p_q), a=1.3962634015954636, v=1.0471975511965976)
      $ 80 "stn2_ref_2_p" "breakAfter"
      set_tcp(p[-3.0E-4,2.5E-4,0.1575,0.0,0.0,0.0])
      movej(get_inverse_kin(pose_trans(stn2_plane, pose_trans(p[.137500819741, -.686313800478, .149495066037, -.008721928164, .022313263547, 3.131433712319], stn2_ref_2_p_p)), qnear=stn2_ref_2_p_q), a=1.3962634015954636, v=1.0471975511965976)
      $ 81 "stn2_ref_3_p" "breakAfter"
      set_tcp(p[-3.0E-4,2.5E-4,0.1575,0.0,0.0,0.0])
      movej(get_inverse_kin(pose_trans(stn2_plane, pose_trans(p[.137500819741, -.686313800478, .149495066037, -.008721928164, .022313263547, 3.131433712319], stn2_ref_3_p_p)), qnear=stn2_ref_3_p_q), a=1.3962634015954636, v=1.0471975511965976)
      $ 82 "stn2_ref_4_p" "breakAfter"
      set_tcp(p[-3.0E-4,2.5E-4,0.1575,0.0,0.0,0.0])
      movej(get_inverse_kin(pose_trans(stn2_plane, pose_trans(p[.137500819741, -.686313800478, .149495066037, -.008721928164, .022313263547, 3.131433712319], stn2_ref_4_p_p)), qnear=stn2_ref_4_p_q), a=1.3962634015954636, v=1.0471975511965976)
      $ 83 "stn2_ref_5_p" "breakAfter"
      set_tcp(p[-3.0E-4,2.5E-4,0.1575,0.0,0.0,0.0])
      movej(get_inverse_kin(pose_trans(stn2_plane, pose_trans(p[.137500819741, -.686313800478, .149495066037, -.008721928164, .022313263547, 3.131433712319], stn2_ref_5_p_p)), qnear=stn2_ref_5_p_q), a=1.3962634015954636, v=1.0471975511965976)
      $ 84 "stn2_ref_6_p" "breakAfter"
      set_tcp(p[-3.0E-4,2.5E-4,0.1575,0.0,0.0,0.0])
      movej(get_inverse_kin(pose_trans(stn2_plane, pose_trans(p[.137500819741, -.686313800478, .149495066037, -.008721928164, .022313263547, 3.131433712319], stn2_ref_6_p_p)), qnear=stn2_ref_6_p_q), a=1.3962634015954636, v=1.0471975511965976)
      $ 85 "'Door positions in subprograms'"
      # 'Door positions in subprograms'
      $ 86 "'Station 3 Reference Positions'"
      # 'Station 3 Reference Positions'
      $ 87 "FahreAchse"
      $ 88 "stn3_home_p" "breakAfter"
      set_tcp(p[-3.0E-4,2.5E-4,0.1575,0.0,0.0,0.0])
      movej(get_inverse_kin(pose_trans(stn3_plane, pose_trans(p[.103513391500, -.760903866624, .250613495596, .000363058783, .000522680433, -.002816727210], stn3_home_p_p)), qnear=stn3_home_p_q), a=1.3962634015954636, v=1.0471975511965976)
      $ 89 "stn3_top_hlp_p" "breakAfter"
      set_tcp(p[-3.0E-4,2.5E-4,0.1575,0.0,0.0,0.0])
      movej(get_inverse_kin(pose_trans(stn3_plane, pose_trans(p[.103513391500, -.760903866624, .250613495596, .000363058783, .000522680433, -.002816727210], stn3_top_hlp_p_p)), qnear=stn3_top_hlp_p_q), a=1.3962634015954636, v=1.0471975511965976)
      $ 90 "stn3_ref_1_p" "breakAfter"
      set_tcp(p[-3.0E-4,2.5E-4,0.1575,0.0,0.0,0.0])
      movej(get_inverse_kin(pose_trans(stn3_plane, pose_trans(p[.103513391500, -.760903866624, .250613495596, .000363058783, .000522680433, -.002816727210], stn3_ref_1_p_p)), qnear=stn3_ref_1_p_q), a=1.3962634015954636, v=1.0471975511965976)
      $ 91 "stn3_ref_2_p" "breakAfter"
      set_tcp(p[-3.0E-4,2.5E-4,0.1575,0.0,0.0,0.0])
      movej(get_inverse_kin(pose_trans(stn3_plane, pose_trans(p[.103513391500, -.760903866624, .250613495596, .000363058783, .000522680433, -.002816727210], stn3_ref_2_p_p)), qnear=stn3_ref_2_p_q), a=1.3962634015954636, v=1.0471975511965976)
      $ 92 "stn3_ref_3_p" "breakAfter"
      set_tcp(p[-3.0E-4,2.5E-4,0.1575,0.0,0.0,0.0])
      movej(get_inverse_kin(pose_trans(stn3_plane, pose_trans(p[.103513391500, -.760903866624, .250613495596, .000363058783, .000522680433, -.002816727210], stn3_ref_3_p_p)), qnear=stn3_ref_3_p_q), a=1.3962634015954636, v=1.0471975511965976)
      $ 93 "stn3_ref_4_p" "breakAfter"
      set_tcp(p[-3.0E-4,2.5E-4,0.1575,0.0,0.0,0.0])
      movej(get_inverse_kin(pose_trans(stn3_plane, pose_trans(p[.103513391500, -.760903866624, .250613495596, .000363058783, .000522680433, -.002816727210], stn3_ref_4_p_p)), qnear=stn3_ref_4_p_q), a=1.3962634015954636, v=1.0471975511965976)
      $ 94 "stn3_ref_5_p" "breakAfter"
      set_tcp(p[-3.0E-4,2.5E-4,0.1575,0.0,0.0,0.0])
      movej(get_inverse_kin(pose_trans(stn3_plane, pose_trans(p[.103513391500, -.760903866624, .250613495596, .000363058783, .000522680433, -.002816727210], stn3_ref_5_p_p)), qnear=stn3_ref_5_p_q), a=1.3962634015954636, v=1.0471975511965976)
      $ 95 "stn3_ref_6_p" "breakAfter"
      set_tcp(p[-3.0E-4,2.5E-4,0.1575,0.0,0.0,0.0])
      movej(get_inverse_kin(pose_trans(stn3_plane, pose_trans(p[.103513391500, -.760903866624, .250613495596, .000363058783, .000522680433, -.002816727210], stn3_ref_6_p_p)), qnear=stn3_ref_6_p_q), a=1.3962634015954636, v=1.0471975511965976)
      $ 96 "stn3_ref_7_p" "breakAfter"
      set_tcp(p[-3.0E-4,2.5E-4,0.1575,0.0,0.0,0.0])
      movej(get_inverse_kin(pose_trans(stn3_plane, pose_trans(p[.103513391500, -.760903866624, .250613495596, .000363058783, .000522680433, -.002816727210], stn3_ref_7_p_p)), qnear=stn3_ref_7_p_q), a=1.3962634015954636, v=1.0471975511965976)
      $ 97 "stn3_ref_8_p" "breakAfter"
      set_tcp(p[-3.0E-4,2.5E-4,0.1575,0.0,0.0,0.0])
      movej(get_inverse_kin(pose_trans(stn3_plane, pose_trans(p[.103513391500, -.760903866624, .250613495596, .000363058783, .000522680433, -.002816727210], stn3_ref_8_p_p)), qnear=stn3_ref_8_p_q), a=1.3962634015954636, v=1.0471975511965976)
      $ 98 "stn3_ini_apr_p" "breakAfter"
      set_tcp(p[-3.0E-4,2.5E-4,0.1575,0.0,0.0,0.0])
      movej(get_inverse_kin(pose_trans(stn3_plane, pose_trans(p[.103513391500, -.760903866624, .250613495596, .000363058783, .000522680433, -.002816727210], stn3_ini_apr_p_p)), qnear=stn3_ini_apr_p_q), a=1.3962634015954636, v=1.0471975511965976)
      $ 99 "stn3_ini_prs_p" "breakAfter"
      set_tcp(p[-3.0E-4,2.5E-4,0.1575,0.0,0.0,0.0])
      movej(get_inverse_kin(pose_trans(stn3_plane, pose_trans(p[.103513391500, -.760903866624, .250613495596, .000363058783, .000522680433, -.002816727210], stn3_ini_prs_p_p)), qnear=stn3_ini_prs_p_q), a=1.3962634015954636, v=1.0471975511965976)
      $ 100 "stn3_apr_run_p" "breakAfter"
      set_tcp(p[-3.0E-4,2.5E-4,0.1575,0.0,0.0,0.0])
      movej(get_inverse_kin(pose_trans(stn3_plane, pose_trans(p[.103513391500, -.760903866624, .250613495596, .000363058783, .000522680433, -.002816727210], stn3_apr_run_p_p)), qnear=stn3_apr_run_p_q), a=1.3962634015954636, v=1.0471975511965976)
      $ 101 "stn3_prss_run_p" "breakAfter"
      set_tcp(p[-3.0E-4,2.5E-4,0.1575,0.0,0.0,0.0])
      movej(get_inverse_kin(pose_trans(stn3_plane, pose_trans(p[.103513391500, -.760903866624, .250613495596, .000363058783, .000522680433, -.002816727210], stn3_prss_run_p_p)), qnear=stn3_prss_run_p_q), a=1.3962634015954636, v=1.0471975511965976)
      $ 102 "'Station 4,6,9,10 reference Positions'"
      # 'Station 4,6,9,10 reference Positions'
      $ 103 "FahreAchse"
      $ 104 "stn6_home_p" "breakAfter"
      set_tcp(p[-3.0E-4,2.5E-4,0.1575,0.0,0.0,0.0])
      movej(get_inverse_kin(pose_trans(stn6_plane, pose_trans(p[.776557109756, -.878329076792, .250244777977, -.001605684562, .009314448336, 1.565629725105], stn6_home_p_p)), qnear=stn6_home_p_q), a=1.3962634015954636, v=1.0471975511965976)
      $ 105 "stn6_help_p" "breakAfter"
      set_tcp(p[-3.0E-4,2.5E-4,0.1575,0.0,0.0,0.0])
      movej(get_inverse_kin(pose_trans(stn6_plane, pose_trans(p[.776557109756, -.878329076792, .250244777977, -.001605684562, .009314448336, 1.565629725105], stn6_help_p_p)), qnear=stn6_help_p_q), a=1.3962634015954636, v=1.0471975511965976)
      $ 106 "stn6_place_p" "breakAfter"
      set_tcp(p[-3.0E-4,2.5E-4,0.1575,0.0,0.0,0.0])
      movej(get_inverse_kin(pose_trans(stn6_plane, pose_trans(p[.776557109756, -.878329076792, .250244777977, -.001605684562, .009314448336, 1.565629725105], stn6_place_p_p)), qnear=stn6_place_p_q), a=1.3962634015954636, v=1.0471975511965976)
      $ 107 "stn4_ref_1_p" "breakAfter"
      set_tcp(p[-3.0E-4,2.5E-4,0.1575,0.0,0.0,0.0])
      movej(get_inverse_kin(pose_trans(stn6_plane, pose_trans(p[.776557109756, -.878329076792, .250244777977, -.001605684562, .009314448336, 1.565629725105], stn4_ref_1_p_p)), qnear=stn4_ref_1_p_q), a=1.3962634015954636, v=1.0471975511965976)
      $ 109 "stn4_cam_help_p" "breakAfter"
      set_tcp(p[-3.0E-4,2.5E-4,0.1575,0.0,0.0,0.0])
      movej(get_inverse_kin(pose_trans(stn6_plane, pose_trans(p[.776557109756, -.878329076792, .250244777977, -.001605684562, .009314448336, 1.565629725105], stn4_cam_help_p_p)), qnear=stn4_cam_help_p_q), a=1.3962634015954636, v=1.0471975511965976)
      $ 110 "stn4_next_hlp_p" "breakAfter"
      set_tcp(p[-3.0E-4,2.5E-4,0.1575,0.0,0.0,0.0])
      movej(get_inverse_kin(pose_trans(stn6_plane, pose_trans(p[.776557109756, -.878329076792, .250244777977, -.001605684562, .009314448336, 1.565629725105], stn4_next_hlp_p_p)), qnear=stn4_next_hlp_p_q), a=1.3962634015954636, v=1.0471975511965976)
      $ 111 "stn5_stn4_hlp_p" "breakAfter"
      set_tcp(p[-3.0E-4,2.5E-4,0.1575,0.0,0.0,0.0])
      movej(get_inverse_kin(pose_trans(stn6_plane, pose_trans(p[.776557109756, -.878329076792, .250244777977, -.001605684562, .009314448336, 1.565629725105], stn5_stn4_hlp_p_p)), qnear=stn5_stn4_hlp_p_q), a=1.3962634015954636, v=1.0471975511965976)
      $ 112 "stn9_dcap_apr_p" "breakAfter"
      set_tcp(p[-3.0E-4,2.5E-4,0.1575,0.0,0.0,0.0])
      movej(get_inverse_kin(pose_trans(stn6_plane, pose_trans(p[.776557109756, -.878329076792, .250244777977, -.001605684562, .009314448336, 1.565629725105], stn9_dcap_apr_p_p)), qnear=stn9_dcap_apr_p_q), a=1.3962634015954636, v=1.0471975511965976)
      $ 113 "stn7_dcap_apr_p" "breakAfter"
      set_tcp(p[-3.0E-4,2.5E-4,0.1575,0.0,0.0,0.0])
      movej(get_inverse_kin(pose_trans(stn6_plane, pose_trans(p[.779413821965, -.869656427631, .149271774994, -.000554336510, .003016566406, 1.568064465904], stn7_dcap_apr_p_p)), qnear=stn7_dcap_apr_p_q), a=1.3962634015954636, v=1.0471975511965976)
      $ 123 "stn10_ref_1_p" "breakAfter"
      set_tcp(p[-3.0E-4,2.5E-4,0.1575,0.0,0.0,0.0])
      movej(get_inverse_kin(pose_trans(stn6_plane, pose_trans(p[.776557109756, -.878329076792, .250244777977, -.001605684562, .009314448336, 1.565629725105], stn10_ref_1_p_p)), qnear=stn10_ref_1_p_q), a=1.3962634015954636, v=1.0471975511965976)
      $ 124 "stn10_ref_2_p" "breakAfter"
      set_tcp(p[-3.0E-4,2.5E-4,0.1575,0.0,0.0,0.0])
      movej(get_inverse_kin(pose_trans(stn6_plane, pose_trans(p[.776557109756, -.878329076792, .250244777977, -.001605684562, .009314448336, 1.565629725105], stn10_ref_2_p_p)), qnear=stn10_ref_2_p_q), a=1.3962634015954636, v=1.0471975511965976)
      $ 125 "stn10_ref_3_p" "breakAfter"
      set_tcp(p[-3.0E-4,2.5E-4,0.1575,0.0,0.0,0.0])
      movej(get_inverse_kin(pose_trans(stn6_plane, pose_trans(p[.776557109756, -.878329076792, .250244777977, -.001605684562, .009314448336, 1.565629725105], stn10_ref_3_p_p)), qnear=stn10_ref_3_p_q), a=1.3962634015954636, v=1.0471975511965976)
      $ 126 "'Station 5 reference Positions'"
      # 'Station 5 reference Positions'
      $ 127 "FahreAchse"
      $ 128 "stn5_rk_rf_1_p" "breakAfter"
      set_tcp(p[-3.0E-4,2.5E-4,0.1575,0.0,0.0,0.0])
      movej(get_inverse_kin(pose_trans(stn5_plane, pose_trans(p[.404793763265, -.880564591570, .218599261998, -.002768907827, .001807604230, 1.568627611983], stn5_rk_rf_1_p_p)), qnear=stn5_rk_rf_1_p_q), a=1.3962634015954636, v=1.0471975511965976)
      $ 129 "stn5_rk_rf_2_p" "breakAfter"
      set_tcp(p[-3.0E-4,2.5E-4,0.1575,0.0,0.0,0.0])
      movej(get_inverse_kin(pose_trans(stn5_plane, pose_trans(p[.404793763265, -.880564591570, .218599261998, -.002768907827, .001807604230, 1.568627611983], stn5_rk_rf_2_p_p)), qnear=stn5_rk_rf_2_p_q), a=1.3962634015954636, v=1.0471975511965976)
      $ 130 "stn5_rk_rf_3_p" "breakAfter"
      set_tcp(p[-3.0E-4,2.5E-4,0.1575,0.0,0.0,0.0])
      movej(get_inverse_kin(pose_trans(stn5_plane, pose_trans(p[.404793763265, -.880564591570, .218599261998, -.002768907827, .001807604230, 1.568627611983], stn5_rk_rf_3_p_p)), qnear=stn5_rk_rf_3_p_q), a=1.3962634015954636, v=1.0471975511965976)
      $ 131 "stn5_tb_rf_1_p" "breakAfter"
      set_tcp(p[-3.0E-4,2.5E-4,0.1575,0.0,0.0,0.0])
      movej(get_inverse_kin(pose_trans(stn5_plane, pose_trans(p[.404793763265, -.880564591570, .218599261998, -.002768907827, .001807604230, 1.568627611983], stn5_tb_rf_1_p_p)), qnear=stn5_tb_rf_1_p_q), a=1.3962634015954636, v=1.0471975511965976)
      $ 132 "stn5_tb_rf_2_p" "breakAfter"
      set_tcp(p[-3.0E-4,2.5E-4,0.1575,0.0,0.0,0.0])
      movej(get_inverse_kin(pose_trans(stn5_plane, pose_trans(p[.404793763265, -.880564591570, .218599261998, -.002768907827, .001807604230, 1.568627611983], stn5_tb_rf_2_p_p)), qnear=stn5_tb_rf_2_p_q), a=1.3962634015954636, v=1.0471975511965976)
      $ 133 "stn5_tb_rf_3_p" "breakAfter"
      set_tcp(p[-3.0E-4,2.5E-4,0.1575,0.0,0.0,0.0])
      movej(get_inverse_kin(pose_trans(stn5_plane, pose_trans(p[.404793763265, -.880564591570, .218599261998, -.002768907827, .001807604230, 1.568627611983], stn5_tb_rf_3_p_p)), qnear=stn5_tb_rf_3_p_q), a=1.3962634015954636, v=1.0471975511965976)
      $ 134 "stn5_tb_rf_4_p" "breakAfter"
      set_tcp(p[-3.0E-4,2.5E-4,0.1575,0.0,0.0,0.0])
      movej(get_inverse_kin(pose_trans(stn5_plane, pose_trans(p[.404793763265, -.880564591570, .218599261998, -.002768907827, .001807604230, 1.568627611983], stn5_tb_rf_4_p_p)), qnear=stn5_tb_rf_4_p_q), a=1.3962634015954636, v=1.0471975511965976)
      $ 135 "stn5_tb_rf_5_p" "breakAfter"
      set_tcp(p[-3.0E-4,2.5E-4,0.1575,0.0,0.0,0.0])
      movej(get_inverse_kin(pose_trans(stn5_plane, pose_trans(p[.404793763265, -.880564591570, .218599261998, -.002768907827, .001807604230, 1.568627611983], stn5_tb_rf_5_p_p)), qnear=stn5_tb_rf_5_p_q), a=1.3962634015954636, v=1.0471975511965976)
      $ 136 "stn5_cw_rf_1_p" "breakAfter"
      set_tcp(p[-3.0E-4,2.5E-4,0.1575,0.0,0.0,0.0])
      movej(get_inverse_kin(pose_trans(stn5_plane, pose_trans(p[.404793763265, -.880564591570, .218599261998, -.002768907827, .001807604230, 1.568627611983], stn5_cw_rf_1_p_p)), qnear=stn5_cw_rf_1_p_q), a=1.3962634015954636, v=1.0471975511965976)
      $ 137 "stn5_cw_rf_2_p" "breakAfter"
      set_tcp(p[-3.0E-4,2.5E-4,0.1575,0.0,0.0,0.0])
      movej(get_inverse_kin(pose_trans(stn5_plane, pose_trans(p[.404793763265, -.880564591570, .218599261998, -.002768907827, .001807604230, 1.568627611983], stn5_cw_rf_2_p_p)), qnear=stn5_cw_rf_2_p_q), a=1.3962634015954636, v=1.0471975511965976)
      $ 138 "'Station 5 init ref Positions'"
      # 'Station 5 init ref Positions'
      $ 152 "'Station 11 reference positions'"
      # 'Station 11 reference positions'
      $ 153 "FahreAchse"
      $ 154 "stn11_home_p" "breakAfter"
      set_tcp(p[-3.0E-4,2.5E-4,0.1575,0.0,0.0,0.0])
      movej(get_inverse_kin(pose_trans(stn6_plane, pose_trans(p[.776557109756, -.878329076792, .250244777977, -.001605684562, .009314448336, 1.565629725105], stn11_home_p_p)), qnear=stn11_home_p_q), a=1.3962634015954636, v=1.0471975511965976)
      $ 155 "stn11_ref_1_p" "breakAfter"
      set_tcp(p[-3.0E-4,2.5E-4,0.1575,0.0,0.0,0.0])
      movej(get_inverse_kin(pose_trans(stn6_plane, pose_trans(p[.776557109756, -.878329076792, .250244777977, -.001605684562, .009314448336, 1.565629725105], stn11_ref_1_p_p)), qnear=stn11_ref_1_p_q), a=1.3962634015954636, v=1.0471975511965976)
      $ 156 "stn11_ref_2_p" "breakAfter"
      set_tcp(p[-3.0E-4,2.5E-4,0.1575,0.0,0.0,0.0])
      movej(get_inverse_kin(pose_trans(stn6_plane, pose_trans(p[.776557109756, -.878329076792, .250244777977, -.001605684562, .009314448336, 1.565629725105], stn11_ref_2_p_p)), qnear=stn11_ref_2_p_q), a=1.3962634015954636, v=1.0471975511965976)
      $ 157 "stn11_ref_3_p" "breakAfter"
      set_tcp(p[-3.0E-4,2.5E-4,0.1575,0.0,0.0,0.0])
      movej(get_inverse_kin(pose_trans(stn6_plane, pose_trans(p[.776557109756, -.878329076792, .250244777977, -.001605684562, .009314448336, 1.565629725105], stn11_ref_3_p_p)), qnear=stn11_ref_3_p_q), a=1.3962634015954636, v=1.0471975511965976)
      $ 158 "stn11_ref_4_p" "breakAfter"
      set_tcp(p[-3.0E-4,2.5E-4,0.1575,0.0,0.0,0.0])
      movej(get_inverse_kin(pose_trans(stn6_plane, pose_trans(p[.776557109756, -.878329076792, .250244777977, -.001605684562, .009314448336, 1.565629725105], stn11_ref_4_p_p)), qnear=stn11_ref_4_p_q), a=1.3962634015954636, v=1.0471975511965976)
      $ 159 "stn11_ref_5_p" "breakAfter"
      set_tcp(p[-3.0E-4,2.5E-4,0.1575,0.0,0.0,0.0])
      movej(get_inverse_kin(pose_trans(stn6_plane, pose_trans(p[.776557109756, -.878329076792, .250244777977, -.001605684562, .009314448336, 1.565629725105], stn11_ref_5_p_p)), qnear=stn11_ref_5_p_q), a=1.3962634015954636, v=1.0471975511965976)
      $ 160 "stn11_ref_6_p" "breakAfter"
      set_tcp(p[-3.0E-4,2.5E-4,0.1575,0.0,0.0,0.0])
      movej(get_inverse_kin(pose_trans(stn6_plane, pose_trans(p[.776557109756, -.878329076792, .250244777977, -.001605684562, .009314448336, 1.565629725105], stn11_ref_6_p_p)), qnear=stn11_ref_6_p_q), a=1.3962634015954636, v=1.0471975511965976)
      $ 161 "stn11_ref_7_p" "breakAfter"
      set_tcp(p[-3.0E-4,2.5E-4,0.1575,0.0,0.0,0.0])
      movej(get_inverse_kin(pose_trans(stn6_plane, pose_trans(p[.776557109756, -.878329076792, .250244777977, -.001605684562, .009314448336, 1.565629725105], stn11_ref_7_p_p)), qnear=stn11_ref_7_p_q), a=1.3962634015954636, v=1.0471975511965976)
      $ 162 "stn11_ref_8_p" "breakAfter"
      set_tcp(p[-3.0E-4,2.5E-4,0.1575,0.0,0.0,0.0])
      movej(get_inverse_kin(pose_trans(stn6_plane, pose_trans(p[.776557109756, -.878329076792, .250244777977, -.001605684562, .009314448336, 1.565629725105], stn11_ref_8_p_p)), qnear=stn11_ref_8_p_q), a=1.3962634015954636, v=1.0471975511965976)
      $ 163 "stn11_ref_9_p" "breakAfter"
      set_tcp(p[-3.0E-4,2.5E-4,0.1575,0.0,0.0,0.0])
      movej(get_inverse_kin(pose_trans(stn6_plane, pose_trans(p[.776557109756, -.878329076792, .250244777977, -.001605684562, .009314448336, 1.565629725105], stn11_ref_9_p_p)), qnear=stn11_ref_9_p_q), a=1.3962634015954636, v=1.0471975511965976)
      $ 164 "stn11_ref10_p" "breakAfter"
      set_tcp(p[-3.0E-4,2.5E-4,0.1575,0.0,0.0,0.0])
      movej(get_inverse_kin(pose_trans(stn6_plane, pose_trans(p[.776557109756, -.878329076792, .250244777977, -.001605684562, .009314448336, 1.565629725105], stn11_ref10_p_p)), qnear=stn11_ref10_p_q), a=1.3962634015954636, v=1.0471975511965976)
      $ 165 "stn11_ref11_p" "breakAfter"
      set_tcp(p[-3.0E-4,2.5E-4,0.1575,0.0,0.0,0.0])
      movej(get_inverse_kin(pose_trans(stn6_plane, pose_trans(p[.776557109756, -.878329076792, .250244777977, -.001605684562, .009314448336, 1.565629725105], stn11_ref11_p_p)), qnear=stn11_ref11_p_q), a=1.3962634015954636, v=1.0471975511965976)
      $ 166 "stn11_ref12_p" "breakAfter"
      set_tcp(p[-3.0E-4,2.5E-4,0.1575,0.0,0.0,0.0])
      movej(get_inverse_kin(pose_trans(stn6_plane, pose_trans(p[.776557109756, -.878329076792, .250244777977, -.001605684562, .009314448336, 1.565629725105], stn11_ref12_p_p)), qnear=stn11_ref12_p_q), a=1.3962634015954636, v=1.0471975511965976)
      $ 167 "'Station 11 door positions in sub program'"
      # 'Station 11 door positions in sub program'
      $ 168 "'Station 7 reference positions'"
      # 'Station 7 reference positions'
      $ 169 "FahreAchse"
      $ 170 "stn7_home_p" "breakAfter"
      set_tcp(p[-3.0E-4,2.5E-4,0.1575,0.0,0.0,0.0])
      movej(get_inverse_kin(pose_trans(stn7_plane, pose_trans(p[.109811488584, -1.023382701287, -.166619380160, .003048702642, -.008599620441, 2.442192581404], stn7_home_p_p)), qnear=stn7_home_p_q), a=1.3962634015954636, v=1.0471975511965976)
      $ 171 "stn7_ref_1_p" "breakAfter"
      set_tcp(p[-3.0E-4,2.5E-4,0.1575,0.0,0.0,0.0])
      movej(get_inverse_kin(pose_trans(stn7_plane, pose_trans(p[.109811488584, -1.023382701287, -.166619380160, .003048702642, -.008599620441, 2.442192581404], stn7_ref_1_p_p)), qnear=stn7_ref_1_p_q), a=1.3962634015954636, v=1.0471975511965976)
      $ 172 "stn7_ref_2_p" "breakAfter"
      set_tcp(p[-3.0E-4,2.5E-4,0.1575,0.0,0.0,0.0])
      movej(get_inverse_kin(pose_trans(stn7_plane, pose_trans(p[.109811488584, -1.023382701287, -.166619380160, .003048702642, -.008599620441, 2.442192581404], stn7_ref_2_p_p)), qnear=stn7_ref_2_p_q), a=1.3962634015954636, v=1.0471975511965976)
      $ 173 "stn7_ref_4_p" "breakAfter"
      set_tcp(p[-3.0E-4,2.5E-4,0.1575,0.0,0.0,0.0])
      movej(get_inverse_kin(pose_trans(stn7_plane, pose_trans(p[.109811488584, -1.023382701287, -.166619380160, .003048702642, -.008599620441, 2.442192581404], stn7_ref_4_p_p)), qnear=stn7_ref_4_p_q), a=1.3962634015954636, v=1.0471975511965976)
      $ 174 "stn7_ref_5_p" "breakAfter"
      set_tcp(p[-3.0E-4,2.5E-4,0.1575,0.0,0.0,0.0])
      movej(get_inverse_kin(pose_trans(stn7_plane, pose_trans(p[.109811488584, -1.023382701287, -.166619380160, .003048702642, -.008599620441, 2.442192581404], stn7_ref_5_p_p)), qnear=stn7_ref_5_p_q), a=1.3962634015954636, v=1.0471975511965976)
      $ 175 "stn7_bin_help_p" "breakAfter"
      set_tcp(p[-3.0E-4,2.5E-4,0.1575,0.0,0.0,0.0])
      movej(get_inverse_kin(pose_trans(stn7_plane, pose_trans(p[.109811488584, -1.023382701287, -.166619380160, .003048702642, -.008599620441, 2.442192581404], stn7_bin_help_p_p)), qnear=stn7_bin_help_p_q), a=1.3962634015954636, v=1.0471975511965976)
      $ 176 "stn7_bin_apr_p" "breakAfter"
      set_tcp(p[-3.0E-4,2.5E-4,0.1575,0.0,0.0,0.0])
      movej(get_inverse_kin(pose_trans(stn7_plane, pose_trans(p[.109811488584, -1.023382701287, -.166619380160, .003048702642, -.008599620441, 2.442192581404], stn7_bin_apr_p_p)), qnear=stn7_bin_apr_p_q), a=1.3962634015954636, v=1.0471975511965976)
      $ 177 "stn7_bin_thrw_p" "breakAfter"
      set_tcp(p[-3.0E-4,2.5E-4,0.1575,0.0,0.0,0.0])
      movej(get_inverse_kin(pose_trans(stn7_plane, pose_trans(p[.109811488584, -1.023382701287, -.166619380160, .003048702642, -.008599620441, 2.442192581404], stn7_bin_thrw_p_p)), qnear=stn7_bin_thrw_p_q), a=1.3962634015954636, v=1.0471975511965976)
      $ 178 "'Station 7 init positions in sub program'"
      # 'Station 7 init positions in sub program'
      $ 179 "'Station 8 reference positions'"
      # 'Station 8 reference positions'
      $ 180 "FahreAchse"
      $ 181 "stn14_stn8_hl_p" "breakAfter"
      set_tcp(p[-3.0E-4,2.5E-4,0.1575,0.0,0.0,0.0])
      movej(get_inverse_kin(pose_trans(stn6_plane, pose_trans(p[.776557109756, -.878329076792, .250244777977, -.001605684562, .009314448336, 1.565629725105], stn14_stn8_hl_p_p)), qnear=stn14_stn8_hl_p_q), a=1.3962634015954636, v=1.0471975511965976)
      $ 182 "stn8_home_p" "breakAfter"
      set_tcp(p[-3.0E-4,2.5E-4,0.1575,0.0,0.0,0.0])
      movej(get_inverse_kin(pose_trans(stn6_plane, pose_trans(p[.776557109756, -.878329076792, .250244777977, -.001605684562, .009314448336, 1.565629725105], stn8_home_p_p)), qnear=stn8_home_p_q), a=1.3962634015954636, v=1.0471975511965976)
      $ 183 "stn8_pl_apr1_p" "breakAfter"
      set_tcp(p[-3.0E-4,2.5E-4,0.1575,0.0,0.0,0.0])
      movej(get_inverse_kin(pose_trans(stn6_plane, pose_trans(p[.776557109756, -.878329076792, .250244777977, -.001605684562, .009314448336, 1.565629725105], stn8_pl_apr1_p_p)), qnear=stn8_pl_apr1_p_q), a=1.3962634015954636, v=1.0471975511965976)
      $ 184 "stn8_pl_apr2_p" "breakAfter"
      set_tcp(p[-3.0E-4,2.5E-4,0.1575,0.0,0.0,0.0])
      movej(get_inverse_kin(pose_trans(stn6_plane, pose_trans(p[.776557109756, -.878329076792, .250244777977, -.001605684562, .009314448336, 1.565629725105], stn8_pl_apr2_p_p)), qnear=stn8_pl_apr2_p_q), a=1.3962634015954636, v=1.0471975511965976)
      $ 185 "stn8_place_p" "breakAfter"
      set_tcp(p[-3.0E-4,2.5E-4,0.1575,0.0,0.0,0.0])
      movej(get_inverse_kin(pose_trans(stn6_plane, pose_trans(p[.776557109756, -.878329076792, .250244777977, -.001605684562, .009314448336, 1.565629725105], stn8_place_p_p)), qnear=stn8_place_p_q), a=1.3962634015954636, v=1.0471975511965976)
      $ 186 "'Station 14 reference positions'"
      # 'Station 14 reference positions'
      $ 187 "FahreAchse"
      $ 188 "stn14_home_p" "breakAfter"
      set_tcp(p[-3.0E-4,2.5E-4,0.1575,0.0,0.0,0.0])
      movej(get_inverse_kin(pose_trans(stn6_plane, pose_trans(p[.779413821965, -.869656427631, .149271774994, -.000554336510, .003016566406, 1.568064465904], stn14_home_p_p)), qnear=stn14_home_p_q), a=1.3962634015954636, v=1.0471975511965976)
      $ 189 "stn14_pk_rk_p" "breakAfter"
      set_tcp(p[-3.0E-4,2.5E-4,0.1575,0.0,0.0,0.0])
      movej(get_inverse_kin(pose_trans(stn6_plane, pose_trans(p[.776557109756, -.878329076792, .250244777977, -.001605684562, .009314448336, 1.565629725105], stn14_pk_rk_p_p)), qnear=stn14_pk_rk_p_q), a=1.3962634015954636, v=1.0471975511965976)
      $ 190 "stn14_pkrk_up_p" "breakAfter"
      set_tcp(p[-3.0E-4,2.5E-4,0.1575,0.0,0.0,0.0])
      movej(get_inverse_kin(pose_trans(stn6_plane, pose_trans(p[.776557109756, -.878329076792, .250244777977, -.001605684562, .009314448336, 1.565629725105], stn14_pkrk_up_p_p)), qnear=stn14_pkrk_up_p_q), a=1.3962634015954636, v=1.0471975511965976)
      $ 191 "stn14_pl_rk_h_p" "breakAfter"
      set_tcp(p[-3.0E-4,2.5E-4,0.1575,0.0,0.0,0.0])
      movej(get_inverse_kin(pose_trans(stn6_plane, pose_trans(p[.776557109756, -.878329076792, .250244777977, -.001605684562, .009314448336, 1.565629725105], stn14_pl_rk_h_p_p)), qnear=stn14_pl_rk_h_p_q), a=1.3962634015954636, v=1.0471975511965976)
      $ 192 "stn14_pl_rk_p" "breakAfter"
      set_tcp(p[-3.0E-4,2.5E-4,0.1575,0.0,0.0,0.0])
      movej(get_inverse_kin(pose_trans(stn6_plane, pose_trans(p[.776557109756, -.878329076792, .250244777977, -.001605684562, .009314448336, 1.565629725105], stn14_pl_rk_p_p)), qnear=stn14_pl_rk_p_q), a=1.3962634015954636, v=1.0471975511965976)
      $ 193 "stn14_plrk_rt_p" "breakAfter"
      set_tcp(p[-3.0E-4,2.5E-4,0.1575,0.0,0.0,0.0])
      movej(get_inverse_kin(pose_trans(stn6_plane, pose_trans(p[.776557109756, -.878329076792, .250244777977, -.001605684562, .009314448336, 1.565629725105], stn14_plrk_rt_p_p)), qnear=stn14_plrk_rt_p_q), a=1.3962634015954636, v=1.0471975511965976)
      $ 194 "stn14_lv_rk_p" "breakAfter"
      set_tcp(p[-3.0E-4,2.5E-4,0.1575,0.0,0.0,0.0])
      movej(get_inverse_kin(pose_trans(stn6_plane, pose_trans(p[.779413821965, -.869656427631, .149271774994, -.000554336510, .003016566406, 1.568064465904], stn14_lv_rk_p_p)), qnear=stn14_lv_rk_p_q), a=1.3962634015954636, v=1.0471975511965976)
      $ 195 "stn14_pl_tb_h_p" "breakAfter"
      set_tcp(p[-3.0E-4,2.5E-4,0.1575,0.0,0.0,0.0])
      movej(get_inverse_kin(pose_trans(stn6_plane, pose_trans(p[.779413821965, -.869656427631, .149271774994, -.000554336510, .003016566406, 1.568064465904], stn14_pl_tb_h_p_p)), qnear=stn14_pl_tb_h_p_q), a=1.3962634015954636, v=1.0471975511965976)
      $ 196 "stn14_ref_1_p" "breakAfter"
      set_tcp(p[-3.0E-4,2.5E-4,0.1575,0.0,0.0,0.0])
      movej(get_inverse_kin(pose_trans(stn6_plane, pose_trans(p[.776557109756, -.878329076792, .250244777977, -.001605684562, .009314448336, 1.565629725105], stn14_ref_1_p_p)), qnear=stn14_ref_1_p_q), a=1.3962634015954636, v=1.0471975511965976)
      $ 197 "stn14_ref_3_p" "breakAfter"
      set_tcp(p[-3.0E-4,2.5E-4,0.1575,0.0,0.0,0.0])
      movej(get_inverse_kin(pose_trans(stn6_plane, pose_trans(p[.776557109756, -.878329076792, .250244777977, -.001605684562, .009314448336, 1.565629725105], stn14_ref_3_p_p)), qnear=stn14_ref_3_p_q), a=1.3962634015954636, v=1.0471975511965976)
      $ 198 "'Station 15 ref positions'"
      # 'Station 15 ref positions'
      $ 199 "FahreAchse"
      $ 200 "stn15_home_p" "breakAfter"
      set_tcp(p[-3.0E-4,2.5E-4,0.1575,0.0,0.0,0.0])
      movej(get_inverse_kin(pose_trans(stn6_plane, pose_trans(p[.776557109756, -.878329076792, .250244777977, -.001605684562, .009314448336, 1.565629725105], stn15_home_p_p)), qnear=stn15_home_p_q), a=1.3962634015954636, v=1.0471975511965976)
      $ 201 "stn15_ref_1_p" "breakAfter"
      set_tcp(p[-3.0E-4,2.5E-4,0.1575,0.0,0.0,0.0])
      movej(get_inverse_kin(pose_trans(stn6_plane, pose_trans(p[.776557109756, -.878329076792, .250244777977, -.001605684562, .009314448336, 1.565629725105], stn15_ref_1_p_p)), qnear=stn15_ref_1_p_q), a=1.3962634015954636, v=1.0471975511965976)
      $ 202 "stn15_ref_2_p" "breakAfter"
      set_tcp(p[-3.0E-4,2.5E-4,0.1575,0.0,0.0,0.0])
      movej(get_inverse_kin(pose_trans(stn6_plane, pose_trans(p[.776557109756, -.878329076792, .250244777977, -.001605684562, .009314448336, 1.565629725105], stn15_ref_2_p_p)), qnear=stn15_ref_2_p_q), a=1.3962634015954636, v=1.0471975511965976)
      $ 203 "stn15_ref_3_p" "breakAfter"
      set_tcp(p[-3.0E-4,2.5E-4,0.1575,0.0,0.0,0.0])
      movej(get_inverse_kin(pose_trans(stn6_plane, pose_trans(p[.776557109756, -.878329076792, .250244777977, -.001605684562, .009314448336, 1.565629725105], stn15_ref_3_p_p)), qnear=stn15_ref_3_p_q), a=1.3962634015954636, v=1.0471975511965976)
    end
    $ 204 "If init_qMast ≟  True "
    if (init_qMast  ==    True  ):
      $ 205 "stn1_ref_1_plan≔pose_trans(pose_inv(stn1_plane), stn1_ref_1_p)"
      global stn1_ref_1_plan= pose_trans ( pose_inv (stn1_plane), pose_trans(stn1_plane, pose_trans(p[.053539610991, -.984987293150, -.024848236577, .000189536594, .000276418508, 3.136265531618], stn1_ref_1_p_p)))
      $ 206 "stn1_ref_2_plan≔pose_trans(pose_inv(stn1_plane), stn1_ref_2_p)"
      global stn1_ref_2_plan= pose_trans ( pose_inv (stn1_plane), pose_trans(stn1_plane, pose_trans(p[.053539610991, -.984987293150, -.024848236577, .000189536594, .000276418508, 3.136265531618], stn1_ref_2_p_p)))
      $ 207 "stn1_ref_3_plan≔pose_trans(pose_inv(stn1_plane), stn1_ref_3_p)"
      global stn1_ref_3_plan= pose_trans ( pose_inv (stn1_plane), pose_trans(stn1_plane, pose_trans(p[.053539610991, -.984987293150, -.024848236577, .000189536594, .000276418508, 3.136265531618], stn1_ref_3_p_p)))
      $ 208 "stn2_rf_1_plane≔pose_trans(pose_inv(stn2_plane), stn2_ref_1_p)"
      global stn2_rf_1_plane= pose_trans ( pose_inv (stn2_plane), pose_trans(stn2_plane, pose_trans(p[.137500819741, -.686313800478, .149495066037, -.008721928164, .022313263547, 3.131433712319], stn2_ref_1_p_p)))
      $ 209 "stn2_rf_2_plane≔pose_trans(pose_inv(stn2_plane), stn2_ref_2_p)"
      global stn2_rf_2_plane= pose_trans ( pose_inv (stn2_plane), pose_trans(stn2_plane, pose_trans(p[.137500819741, -.686313800478, .149495066037, -.008721928164, .022313263547, 3.131433712319], stn2_ref_2_p_p)))
      $ 210 "stn2_rf_3_plane≔pose_trans(pose_inv(stn2_plane), stn2_ref_3_p)"
      global stn2_rf_3_plane= pose_trans ( pose_inv (stn2_plane), pose_trans(stn2_plane, pose_trans(p[.137500819741, -.686313800478, .149495066037, -.008721928164, .022313263547, 3.131433712319], stn2_ref_3_p_p)))
      $ 211 "stn2_rf_4_plane≔pose_trans(pose_inv(stn2_plane), stn2_ref_4_p)"
      global stn2_rf_4_plane= pose_trans ( pose_inv (stn2_plane), pose_trans(stn2_plane, pose_trans(p[.137500819741, -.686313800478, .149495066037, -.008721928164, .022313263547, 3.131433712319], stn2_ref_4_p_p)))
      $ 212 "stn2_rf_5_plane≔pose_trans(pose_inv(stn2_plane), stn2_ref_5_p)"
      global stn2_rf_5_plane= pose_trans ( pose_inv (stn2_plane), pose_trans(stn2_plane, pose_trans(p[.137500819741, -.686313800478, .149495066037, -.008721928164, .022313263547, 3.131433712319], stn2_ref_5_p_p)))
      $ 213 "stn2_rf_6_plane≔pose_trans(pose_inv(stn2_plane), stn2_ref_6_p)"
      global stn2_rf_6_plane= pose_trans ( pose_inv (stn2_plane), pose_trans(stn2_plane, pose_trans(p[.137500819741, -.686313800478, .149495066037, -.008721928164, .022313263547, 3.131433712319], stn2_ref_6_p_p)))
      $ 214 "stn3_ref_1_plan≔pose_trans(pose_inv(stn3_plane), stn3_ref_1_p)"
      global stn3_ref_1_plan= pose_trans ( pose_inv (stn3_plane), pose_trans(stn3_plane, pose_trans(p[.103513391500, -.760903866624, .250613495596, .000363058783, .000522680433, -.002816727210], stn3_ref_1_p_p)))
      $ 215 "stn3_ref_2_plan≔pose_trans(pose_inv(stn3_plane), stn3_ref_2_p)"
      global stn3_ref_2_plan= pose_trans ( pose_inv (stn3_plane), pose_trans(stn3_plane, pose_trans(p[.103513391500, -.760903866624, .250613495596, .000363058783, .000522680433, -.002816727210], stn3_ref_2_p_p)))
      $ 216 "stn3_ref_3_plan≔pose_trans(pose_inv(stn3_plane), stn3_ref_3_p)"
      global stn3_ref_3_plan= pose_trans ( pose_inv (stn3_plane), pose_trans(stn3_plane, pose_trans(p[.103513391500, -.760903866624, .250613495596, .000363058783, .000522680433, -.002816727210], stn3_ref_3_p_p)))
      $ 217 "stn3_ref_4_plan≔pose_trans(pose_inv(stn3_plane), stn3_ref_4_p)"
      global stn3_ref_4_plan= pose_trans ( pose_inv (stn3_plane), pose_trans(stn3_plane, pose_trans(p[.103513391500, -.760903866624, .250613495596, .000363058783, .000522680433, -.002816727210], stn3_ref_4_p_p)))
      $ 218 "stn3_ref_5_plan≔pose_trans(pose_inv(stn3_plane), stn3_ref_5_p)"
      global stn3_ref_5_plan= pose_trans ( pose_inv (stn3_plane), pose_trans(stn3_plane, pose_trans(p[.103513391500, -.760903866624, .250613495596, .000363058783, .000522680433, -.002816727210], stn3_ref_5_p_p)))
      $ 219 "stn3_ref_6_plan≔pose_trans(pose_inv(stn3_plane), stn3_ref_6_p)"
      global stn3_ref_6_plan= pose_trans ( pose_inv (stn3_plane), pose_trans(stn3_plane, pose_trans(p[.103513391500, -.760903866624, .250613495596, .000363058783, .000522680433, -.002816727210], stn3_ref_6_p_p)))
      $ 220 "stn3_ref_7_plan≔pose_trans(pose_inv(stn3_plane), stn3_ref_7_p)"
      global stn3_ref_7_plan= pose_trans ( pose_inv (stn3_plane), pose_trans(stn3_plane, pose_trans(p[.103513391500, -.760903866624, .250613495596, .000363058783, .000522680433, -.002816727210], stn3_ref_7_p_p)))
      $ 221 "stn3_ref_8_plan≔pose_trans(pose_inv(stn3_plane), stn3_ref_8_p)"
      global stn3_ref_8_plan= pose_trans ( pose_inv (stn3_plane), pose_trans(stn3_plane, pose_trans(p[.103513391500, -.760903866624, .250613495596, .000363058783, .000522680433, -.002816727210], stn3_ref_8_p_p)))
      $ 222 "stn5_ref_1_plan≔pose_trans(pose_inv(stn5_plane),stn5_tb_rf_1_p)"
      global stn5_ref_1_plan= pose_trans ( pose_inv (stn5_plane),pose_trans(stn5_plane, pose_trans(p[.404793763265, -.880564591570, .218599261998, -.002768907827, .001807604230, 1.568627611983], stn5_tb_rf_1_p_p)))
      $ 223 "stn5_ref_2_plan≔pose_trans(pose_inv(stn5_plane),stn5_tb_rf_2_p)"
      global stn5_ref_2_plan= pose_trans ( pose_inv (stn5_plane),pose_trans(stn5_plane, pose_trans(p[.404793763265, -.880564591570, .218599261998, -.002768907827, .001807604230, 1.568627611983], stn5_tb_rf_2_p_p)))
      $ 224 "stn5_ref_3_plan≔pose_trans(pose_inv(stn5_plane),stn5_tb_rf_3_p)"
      global stn5_ref_3_plan= pose_trans ( pose_inv (stn5_plane),pose_trans(stn5_plane, pose_trans(p[.404793763265, -.880564591570, .218599261998, -.002768907827, .001807604230, 1.568627611983], stn5_tb_rf_3_p_p)))
      $ 225 "stn5_ref_4_plan≔pose_trans(pose_inv(stn5_plane),stn5_tb_rf_4_p)"
      global stn5_ref_4_plan= pose_trans ( pose_inv (stn5_plane),pose_trans(stn5_plane, pose_trans(p[.404793763265, -.880564591570, .218599261998, -.002768907827, .001807604230, 1.568627611983], stn5_tb_rf_4_p_p)))
      $ 226 "stn5_ref_5_plan≔pose_trans(pose_inv(stn5_plane),stn5_tb_rf_5_p)"
      global stn5_ref_5_plan= pose_trans ( pose_inv (stn5_plane),pose_trans(stn5_plane, pose_trans(p[.404793763265, -.880564591570, .218599261998, -.002768907827, .001807604230, 1.568627611983], stn5_tb_rf_5_p_p)))
      $ 227 "stn5_rk_1_plane≔pose_trans(pose_inv(stn5_plane),stn5_rk_rf_1_p)"
      global stn5_rk_1_plane= pose_trans ( pose_inv (stn5_plane),pose_trans(stn5_plane, pose_trans(p[.404793763265, -.880564591570, .218599261998, -.002768907827, .001807604230, 1.568627611983], stn5_rk_rf_1_p_p)))
      $ 228 "stn5_rk_2_plane≔pose_trans(pose_inv(stn5_plane),stn5_rk_rf_2_p)"
      global stn5_rk_2_plane= pose_trans ( pose_inv (stn5_plane),pose_trans(stn5_plane, pose_trans(p[.404793763265, -.880564591570, .218599261998, -.002768907827, .001807604230, 1.568627611983], stn5_rk_rf_2_p_p)))
      $ 229 "stn5_rk_3_plane≔pose_trans(pose_inv(stn5_plane),stn5_rk_rf_3_p)"
      global stn5_rk_3_plane= pose_trans ( pose_inv (stn5_plane),pose_trans(stn5_plane, pose_trans(p[.404793763265, -.880564591570, .218599261998, -.002768907827, .001807604230, 1.568627611983], stn5_rk_rf_3_p_p)))
      $ 230 "stn5_cw_1_plane≔pose_trans(pose_inv(stn5_plane),stn5_cw_rf_1_p)"
      global stn5_cw_1_plane= pose_trans ( pose_inv (stn5_plane),pose_trans(stn5_plane, pose_trans(p[.404793763265, -.880564591570, .218599261998, -.002768907827, .001807604230, 1.568627611983], stn5_cw_rf_1_p_p)))
      $ 231 "stn5_cw_2_plane≔pose_trans(pose_inv(stn5_plane), stn5_cw_rf_2_p)"
      global stn5_cw_2_plane= pose_trans ( pose_inv (stn5_plane), pose_trans(stn5_plane, pose_trans(p[.404793763265, -.880564591570, .218599261998, -.002768907827, .001807604230, 1.568627611983], stn5_cw_rf_2_p_p)))
      $ 232 "stn7_ref_1_plan≔pose_trans(pose_inv(stn7_plane), stn7_ref_1_p)"
      global stn7_ref_1_plan= pose_trans ( pose_inv (stn7_plane), pose_trans(stn7_plane, pose_trans(p[.109811488584, -1.023382701287, -.166619380160, .003048702642, -.008599620441, 2.442192581404], stn7_ref_1_p_p)))
      $ 233 "stn7_ref_2_plan≔pose_trans(pose_inv(stn7_plane), stn7_ref_2_p)"
      global stn7_ref_2_plan= pose_trans ( pose_inv (stn7_plane), pose_trans(stn7_plane, pose_trans(p[.109811488584, -1.023382701287, -.166619380160, .003048702642, -.008599620441, 2.442192581404], stn7_ref_2_p_p)))
      $ 234 "stn7_ref_3_plan≔pose_trans(pose_inv(stn7_plane), stn7_ref_1_p)"
      global stn7_ref_3_plan= pose_trans ( pose_inv (stn7_plane), pose_trans(stn7_plane, pose_trans(p[.109811488584, -1.023382701287, -.166619380160, .003048702642, -.008599620441, 2.442192581404], stn7_ref_1_p_p)))
      $ 235 "stn7_ref_4_plan≔pose_trans(pose_inv(stn7_plane), stn7_ref_4_p)"
      global stn7_ref_4_plan= pose_trans ( pose_inv (stn7_plane), pose_trans(stn7_plane, pose_trans(p[.109811488584, -1.023382701287, -.166619380160, .003048702642, -.008599620441, 2.442192581404], stn7_ref_4_p_p)))
      $ 236 "stn7_ref_5_plan≔pose_trans(pose_inv(stn7_plane), stn7_ref_5_p)"
      global stn7_ref_5_plan= pose_trans ( pose_inv (stn7_plane), pose_trans(stn7_plane, pose_trans(p[.109811488584, -1.023382701287, -.166619380160, .003048702642, -.008599620441, 2.442192581404], stn7_ref_5_p_p)))
      $ 237 "stn10_ref_1_pln≔pose_trans(pose_inv(stn6_plane), stn10_ref_1_p)"
      global stn10_ref_1_pln= pose_trans ( pose_inv (stn6_plane), pose_trans(stn6_plane, pose_trans(p[.776557109756, -.878329076792, .250244777977, -.001605684562, .009314448336, 1.565629725105], stn10_ref_1_p_p)))
      $ 238 "stn10_ref_2_pln≔pose_trans(pose_inv(stn6_plane), stn10_ref_2_p)"
      global stn10_ref_2_pln= pose_trans ( pose_inv (stn6_plane), pose_trans(stn6_plane, pose_trans(p[.776557109756, -.878329076792, .250244777977, -.001605684562, .009314448336, 1.565629725105], stn10_ref_2_p_p)))
      $ 239 "stn10_ref_3_pln≔pose_trans(pose_inv(stn6_plane), stn10_ref_3_p)"
      global stn10_ref_3_pln= pose_trans ( pose_inv (stn6_plane), pose_trans(stn6_plane, pose_trans(p[.776557109756, -.878329076792, .250244777977, -.001605684562, .009314448336, 1.565629725105], stn10_ref_3_p_p)))
      $ 240 "stn11_ref_1_pln≔pose_trans(pose_inv(stn6_plane), stn11_ref_1_p)"
      global stn11_ref_1_pln= pose_trans ( pose_inv (stn6_plane), pose_trans(stn6_plane, pose_trans(p[.776557109756, -.878329076792, .250244777977, -.001605684562, .009314448336, 1.565629725105], stn11_ref_1_p_p)))
      $ 241 "stn11_ref_2_pln≔pose_trans(pose_inv(stn6_plane), stn11_ref_2_p)"
      global stn11_ref_2_pln= pose_trans ( pose_inv (stn6_plane), pose_trans(stn6_plane, pose_trans(p[.776557109756, -.878329076792, .250244777977, -.001605684562, .009314448336, 1.565629725105], stn11_ref_2_p_p)))
      $ 242 "stn11_ref_3_pln≔pose_trans(pose_inv(stn6_plane), stn11_ref_3_p)"
      global stn11_ref_3_pln= pose_trans ( pose_inv (stn6_plane), pose_trans(stn6_plane, pose_trans(p[.776557109756, -.878329076792, .250244777977, -.001605684562, .009314448336, 1.565629725105], stn11_ref_3_p_p)))
      $ 243 "stn11_ref_4_pln≔pose_trans(pose_inv(stn6_plane), stn11_ref_4_p)"
      global stn11_ref_4_pln= pose_trans ( pose_inv (stn6_plane), pose_trans(stn6_plane, pose_trans(p[.776557109756, -.878329076792, .250244777977, -.001605684562, .009314448336, 1.565629725105], stn11_ref_4_p_p)))
      $ 244 "stn11_ref_5_pln≔pose_trans(pose_inv(stn6_plane), stn11_ref_5_p)"
      global stn11_ref_5_pln= pose_trans ( pose_inv (stn6_plane), pose_trans(stn6_plane, pose_trans(p[.776557109756, -.878329076792, .250244777977, -.001605684562, .009314448336, 1.565629725105], stn11_ref_5_p_p)))
      $ 245 "stn11_ref_6_pln≔pose_trans(pose_inv(stn6_plane), stn11_ref_6_p)"
      global stn11_ref_6_pln= pose_trans ( pose_inv (stn6_plane), pose_trans(stn6_plane, pose_trans(p[.776557109756, -.878329076792, .250244777977, -.001605684562, .009314448336, 1.565629725105], stn11_ref_6_p_p)))
      $ 246 "stn11_ref_7_pln≔pose_trans(pose_inv(stn6_plane), stn11_ref_7_p)"
      global stn11_ref_7_pln= pose_trans ( pose_inv (stn6_plane), pose_trans(stn6_plane, pose_trans(p[.776557109756, -.878329076792, .250244777977, -.001605684562, .009314448336, 1.565629725105], stn11_ref_7_p_p)))
      $ 247 "stn11_ref_8_pln≔pose_trans(pose_inv(stn6_plane), stn11_ref_8_p)"
      global stn11_ref_8_pln= pose_trans ( pose_inv (stn6_plane), pose_trans(stn6_plane, pose_trans(p[.776557109756, -.878329076792, .250244777977, -.001605684562, .009314448336, 1.565629725105], stn11_ref_8_p_p)))
      $ 248 "stn11_ref_9_pln≔pose_trans(pose_inv(stn6_plane), stn11_ref_9_p)"
      global stn11_ref_9_pln= pose_trans ( pose_inv (stn6_plane), pose_trans(stn6_plane, pose_trans(p[.776557109756, -.878329076792, .250244777977, -.001605684562, .009314448336, 1.565629725105], stn11_ref_9_p_p)))
      $ 249 "stn11_ref_10_pl≔pose_trans(pose_inv(stn6_plane), stn11_ref10_p)"
      global stn11_ref_10_pl= pose_trans ( pose_inv (stn6_plane), pose_trans(stn6_plane, pose_trans(p[.776557109756, -.878329076792, .250244777977, -.001605684562, .009314448336, 1.565629725105], stn11_ref10_p_p)))
      $ 250 "stn11_ref_11_pl≔pose_trans(pose_inv(stn6_plane), stn11_ref11_p)"
      global stn11_ref_11_pl= pose_trans ( pose_inv (stn6_plane), pose_trans(stn6_plane, pose_trans(p[.776557109756, -.878329076792, .250244777977, -.001605684562, .009314448336, 1.565629725105], stn11_ref11_p_p)))
      $ 251 "stn11_ref_12_pl≔pose_trans(pose_inv(stn6_plane), stn11_ref12_p)"
      global stn11_ref_12_pl= pose_trans ( pose_inv (stn6_plane), pose_trans(stn6_plane, pose_trans(p[.776557109756, -.878329076792, .250244777977, -.001605684562, .009314448336, 1.565629725105], stn11_ref12_p_p)))
      $ 252 "stn14_ref_1_pln≔pose_trans(pose_inv(stn6_plane), stn14_ref_1_p)"
      global stn14_ref_1_pln= pose_trans ( pose_inv (stn6_plane), pose_trans(stn6_plane, pose_trans(p[.776557109756, -.878329076792, .250244777977, -.001605684562, .009314448336, 1.565629725105], stn14_ref_1_p_p)))
      $ 253 "stn14_ref_3_pln≔pose_trans(pose_inv(stn6_plane), stn14_ref_3_p)"
      global stn14_ref_3_pln= pose_trans ( pose_inv (stn6_plane), pose_trans(stn6_plane, pose_trans(p[.776557109756, -.878329076792, .250244777977, -.001605684562, .009314448336, 1.565629725105], stn14_ref_3_p_p)))
      $ 254 "stn15_ref_1_pln≔pose_trans(pose_inv(stn6_plane), stn15_ref_1_p)"
      global stn15_ref_1_pln= pose_trans ( pose_inv (stn6_plane), pose_trans(stn6_plane, pose_trans(p[.776557109756, -.878329076792, .250244777977, -.001605684562, .009314448336, 1.565629725105], stn15_ref_1_p_p)))
      $ 255 "stn15_ref_2_pln≔pose_trans(pose_inv(stn6_plane), stn15_ref_2_p)"
      global stn15_ref_2_pln= pose_trans ( pose_inv (stn6_plane), pose_trans(stn6_plane, pose_trans(p[.776557109756, -.878329076792, .250244777977, -.001605684562, .009314448336, 1.565629725105], stn15_ref_2_p_p)))
      $ 256 "stn15_ref_3_pln≔pose_trans(pose_inv(stn6_plane), stn15_ref_3_p)"
      global stn15_ref_3_pln= pose_trans ( pose_inv (stn6_plane), pose_trans(stn6_plane, pose_trans(p[.776557109756, -.878329076792, .250244777977, -.001605684562, .009314448336, 1.565629725105], stn15_ref_3_p_p)))
      $ 257 "qMast.reset()"
      qMast.reset()
      $ 258 "qMast.init_q400()"
      qMast.init_q400()
      $ 259 "qMast.set_stn1_grid(1,stn1_ref_1_plan,stn1_ref_2_plan,stn1_ref_3_plan,stn1_rows,stn1_cols)"
      qMast.set_stn1_grid(1,stn1_ref_1_plan,stn1_ref_2_plan,stn1_ref_3_plan,stn1_rows,stn1_cols)
      $ 260 "qMast.set_stn2_grid(1,stn2_rf_1_plane,stn2_rf_2_plane,stn2_rf_3_plane,stn2_rf_4_plane,stn2_rf_5_plane,stn2_rf_6_plane)"
      qMast.set_stn2_grid(1,stn2_rf_1_plane,stn2_rf_2_plane,stn2_rf_3_plane,stn2_rf_4_plane,stn2_rf_5_plane,stn2_rf_6_plane)
      $ 261 "qMast.set_stn3_grid(1, stn3_ref_1_plan, stn3_ref_2_plan, stn3_ref_3_plan, stn3_ref_4_plan, stn3_ref_5_plan, stn3_ref_6_plan, stn3_ref_7_plan, stn3_ref_8_plan)"
      qMast.set_stn3_grid(1, stn3_ref_1_plan, stn3_ref_2_plan, stn3_ref_3_plan, stn3_ref_4_plan, stn3_ref_5_plan, stn3_ref_6_plan, stn3_ref_7_plan, stn3_ref_8_plan)
      $ 262 "qMast.set_stn5_grid(1,stn5_ref_1_plan,stn5_ref_2_plan,stn5_ref_3_plan,stn5_rows_parnt,stn5_cols_parnt,stn5_ref_4_plan,stn5_ref_5_plan,stn5_rows_child,stn5_cols_child)"
      qMast.set_stn5_grid(1,stn5_ref_1_plan,stn5_ref_2_plan,stn5_ref_3_plan,stn5_rows_parnt,stn5_cols_parnt,stn5_ref_4_plan,stn5_ref_5_plan,stn5_rows_child,stn5_cols_child)
      $ 263 "qMast.set_stn5_counter_grid(stn5_cw_1_plane, stn5_cw_2_plane)"
      qMast.set_stn5_counter_grid(stn5_cw_1_plane, stn5_cw_2_plane)
      $ 264 "qMast.set_stn5_batch_grid(1,stn5_rk_1_plane,stn5_rk_2_plane,stn5_rk_3_plane,4,2)"
      qMast.set_stn5_batch_grid(1,stn5_rk_1_plane,stn5_rk_2_plane,stn5_rk_3_plane,4,2)
      $ 265 "qMast.set_stn7_grid(1,stn7_ref_1_plan,stn7_ref_2_plan,stn7_ref_3_plan,stn7_rows_parnt,stn7_cols_parnt,stn7_ref_4_plan,stn7_ref_5_plan,stn7_rows_child,stn7_cols_child)"
      qMast.set_stn7_grid(1,stn7_ref_1_plan,stn7_ref_2_plan,stn7_ref_3_plan,stn7_rows_parnt,stn7_cols_parnt,stn7_ref_4_plan,stn7_ref_5_plan,stn7_rows_child,stn7_cols_child)
      $ 266 "qMast.set_stn10_grid(1,stn10_ref_1_pln,stn10_ref_2_pln,stn10_ref_3_pln,8,4)"
      qMast.set_stn10_grid(1,stn10_ref_1_pln,stn10_ref_2_pln,stn10_ref_3_pln,8,4)
      $ 267 "qMast.set_stn11_grid(1,stn11_ref_1_pln,stn11_ref_2_pln,stn11_ref_3_pln,stn11_ref_4_pln,stn11_ref_5_pln,stn11_ref_6_pln,stn11_ref_7_pln,stn11_ref_8_pln,stn11_ref_9_pln,stn11_ref_10_pl,stn11_ref_11_pl,stn11_ref_12_pl,8,4)"
      qMast.set_stn11_grid(1,stn11_ref_1_pln,stn11_ref_2_pln,stn11_ref_3_pln,stn11_ref_4_pln,stn11_ref_5_pln,stn11_ref_6_pln,stn11_ref_7_pln,stn11_ref_8_pln,stn11_ref_9_pln,stn11_ref_10_pl,stn11_ref_11_pl,stn11_ref_12_pl,8,4)
      $ 268 "qMast.set_stn14_grid(1,stn14_ref_1_pln,stn14_ref_1_pln,stn14_ref_3_pln,5,1)"
      qMast.set_stn14_grid(1,stn14_ref_1_pln,stn14_ref_1_pln,stn14_ref_3_pln,5,1)
      $ 269 "qMast.set_stn15_grid(1,stn15_ref_1_pln,stn15_ref_2_pln,stn15_ref_3_pln,8,4)"
      qMast.set_stn15_grid(1,stn15_ref_1_pln,stn15_ref_2_pln,stn15_ref_3_pln,8,4)
      # begin: URCap Program Node
      #   Source: Robotiq_Grippers, 1.8.13.22852, Robotiq Inc.
      #   Type: Greifer aktivieren
      $ 270 "Greifer zurücksetzen und aktivieren"

      kill rq_gripper_communication_thread
      rq_gripper_communication_thread_started = False
      rq_close_gripper_socket("1")
      rq_close_gripper_socket("2")
      rq_close_gripper_socket("3")
      rq_close_gripper_socket("4")

      rq_init_comm_if_connected(9, "1")
      rq_init_comm_if_connected(2, "2")
      rq_init_comm_if_connected(3, "3")
      rq_init_comm_if_connected(4, "4")
      rq_print_connected_grippers()
      rq_gripper_communication_thread = run rq_gripper_communication()

      while(not rq_gripper_communication_thread_started):
          sleep(0.008)
      end

      rq_set_max_current_for_all_grippers()

      reset_and_activate = True

